LIN {X 0.262,Y -671.425,Z 418.419,A 0.000,B 0.000,C 90.000,E1 291.408} C_DIS
LIN {X -0.297,Y -673.117,Z 418.412,A 0.000,B 0.000,C 90.000,E1 290.248} C_DIS
LIN {X -0.129,Y -673.902,Z 418.407,A 0.000,B 0.000,C 90.000,E1 289.268} C_DIS
LIN {X -0.108,Y -674.468,Z 418.403,A 0.000,B 0.000,C 90.000,E1 288.544} C_DIS
LIN {X 0.005,Y -675.043,Z 418.396,A 0.000,B 0.000,C 90.000,E1 287.330} C_DIS
LIN {X -0.218,Y -675.211,Z 418.391,A 0.000,B 0.000,C 90.000,E1 286.386} C_DIS
LIN {X -0.297,Y -675.251,Z 418.384,A 0.000,B 0.000,C 90.000,E1 285.190} C_DIS
LIN {X 0.102,Y -675.047,Z 418.378,A 0.000,B 0.000,C 90.000,E1 283.953} C_DIS
LIN {X -0.211,Y -674.521,Z 418.370,A 0.000,B 0.000,C 90.000,E1 282.535} C_DIS
LIN {X -0.024,Y -673.626,Z 418.362,A 0.000,B 0.000,C 90.000,E1 281.074} C_DIS
LIN {X 0.207,Y -672.646,Z 418.355,A 0.000,B 0.000,C 90.000,E1 279.849} C_DIS
LIN {X 0.235,Y -671.359,Z 418.347,A 0.000,B 0.000,C 90.000,E1 278.398} C_DIS
LIN {X -0.033,Y -669.490,Z 418.336,A 0.000,B 0.000,C 90.000,E1 276.486} C_DIS
LIN {X -0.069,Y -668.227,Z 418.329,A 0.000,B 0.000,C 90.000,E1 275.277} C_DIS
LIN {X -0.176,Y -666.863,Z 418.323,A 0.000,B 0.000,C 90.000,E1 274.073} C_DIS
LIN {X -0.258,Y -665.172,Z 418.316,A 0.000,B 0.000,C 90.000,E1 272.865} C_DIS
LIN {X -0.263,Y -663.871,Z 418.310,A 0.000,B 0.000,C 90.000,E1 271.892} C_DIS
LIN {X 0.052,Y -661.562,Z 418.302,A 0.000,B 0.000,C 90.000,E1 270.401} C_DIS
LIN {X -0.174,Y -659.257,Z 418.296,A 0.000,B 0.000,C 90.000,E1 269.198} C_DIS
LIN {X 0.235,Y -656.673,Z 418.289,A 0.000,B 0.000,C 90.000,E1 267.936} C_DIS
LIN {X -0.252,Y -653.217,Z 418.280,A 0.000,B 0.000,C 90.000,E1 266.502} C_DIS
LIN {X -0.115,Y -649.497,Z 418.272,A 0.000,B 0.000,C 90.000,E1 265.008} C_DIS
LIN {X 0.172,Y -646.188,Z 418.265,A 0.000,B 0.000,C 90.000,E1 263.742} C_DIS
LIN {X -0.163,Y -642.674,Z 418.258,A 0.000,B 0.000,C 90.000,E1 262.527} C_DIS
LIN {X 0.085,Y -638.920,Z 418.251,A 0.000,B 0.000,C 90.000,E1 261.254} C_DIS
LIN {X 0.257,Y -635.010,Z 418.245,A 0.000,B 0.000,C 90.000,E1 259.982} C_DIS
LIN {X -0.157,Y -631.024,Z 418.238,A 0.000,B 0.000,C 90.000,E1 258.757} C_DIS
LIN {X 0.308,Y -627.809,Z 418.232,A 0.000,B 0.000,C 90.000,E1 257.701} C_DIS
LIN {X 0.311,Y -622.852,Z 418.223,A 0.000,B 0.000,C 90.000,E1 256.172} C_DIS
LIN {X 0.052,Y -619.414,Z 418.218,A 0.000,B 0.000,C 90.000,E1 255.172} C_DIS
LIN {X -0.325,Y -614.936,Z 418.211,A 0.000,B 0.000,C 90.000,E1 253.921} C_DIS
LIN {X -0.260,Y -609.408,Z 418.202,A 0.000,B 0.000,C 90.000,E1 252.362} C_DIS
LIN {X -0.042,Y -604.626,Z 418.195,A 0.000,B 0.000,C 90.000,E1 251.040} C_DIS
LIN {X 0.199,Y -598.715,Z 418.186,A 0.000,B 0.000,C 90.000,E1 249.444} C_DIS
LIN {X -0.036,Y -594.599,Z 418.180,A 0.000,B 0.000,C 90.000,E1 248.411} C_DIS
LIN {X -0.110,Y -590.373,Z 418.174,A 0.000,B 0.000,C 90.000,E1 247.358} C_DIS
LIN {X 0.174,Y -584.953,Z 418.167,A 0.000,B 0.000,C 90.000,E1 245.997} C_DIS
LIN {X 0.064,Y -579.379,Z 418.159,A 0.000,B 0.000,C 90.000,E1 244.665} C_DIS
LIN {X -0.191,Y -571.625,Z 418.149,A 0.000,B 0.000,C 90.000,E1 242.794} C_DIS
LIN {X 0.055,Y -564.970,Z 418.140,A 0.000,B 0.000,C 90.000,E1 241.129} C_DIS
LIN {X 0.206,Y -558.507,Z 418.130,A 0.000,B 0.000,C 90.000,E1 239.459} C_DIS
LIN {X 0.046,Y -550.141,Z 418.118,A 0.000,B 0.000,C 90.000,E1 237.248} C_DIS
LIN {X -0.278,Y -544.124,Z 418.109,A 0.000,B 0.000,C 90.000,E1 235.595} C_DIS
LIN {X 0.018,Y -538.215,Z 418.099,A 0.000,B 0.000,C 90.000,E1 233.863} C_DIS
LIN {X 0.059,Y -533.367,Z 418.091,A 0.000,B 0.000,C 90.000,E1 232.431} C_DIS
LIN {X -0.095,Y -527.441,Z 418.082,A 0.000,B 0.000,C 90.000,E1 230.723} C_DIS
LIN {X 0.096,Y -518.241,Z 418.066,A 0.000,B 0.000,C 90.000,E1 227.796} C_DIS
LIN {X 0.015,Y -513.892,Z 418.057,A 0.000,B 0.000,C 90.000,E1 226.338} C_DIS
LIN {X -0.240,Y -508.752,Z 418.048,A 0.000,B 0.000,C 90.000,E1 224.595} C_DIS
LIN {X 0.108,Y -503.657,Z 418.038,A 0.000,B 0.000,C 90.000,E1 222.771} C_DIS
LIN {X -0.137,Y -497.952,Z 418.026,A 0.000,B 0.000,C 90.000,E1 220.701} C_DIS
LIN {X -0.011,Y -493.110,Z 418.016,A 0.000,B 0.000,C 90.000,E1 218.874} C_DIS
LIN {X 0.156,Y -488.555,Z 418.006,A 0.000,B 0.000,C 90.000,E1 217.030} C_DIS
LIN {X -0.121,Y -482.585,Z 417.992,A 0.000,B 0.000,C 90.000,E1 214.612} C_DIS
LIN {X -0.060,Y -478.327,Z 417.982,A 0.000,B 0.000,C 90.000,E1 212.752} C_DIS
LIN {X -0.138,Y -474.780,Z 417.973,A 0.000,B 0.000,C 90.000,E1 211.209} C_DIS
LIN {X 0.056,Y -469.855,Z 417.961,A 0.000,B 0.000,C 90.000,E1 208.999} C_DIS
LIN {X -0.016,Y -466.300,Z 417.952,A 0.000,B 0.000,C 90.000,E1 207.436} C_DIS
LIN {X 0.095,Y -461.208,Z 417.940,A 0.000,B 0.000,C 90.000,E1 205.207} C_DIS
LIN {X -0.128,Y -457.419,Z 417.931,A 0.000,B 0.000,C 90.000,E1 203.643} C_DIS
LIN {X -0.101,Y -452.986,Z 417.921,A 0.000,B 0.000,C 90.000,E1 201.716} C_DIS
LIN {X 0.121,Y -446.616,Z 417.904,A 0.000,B 0.000,C 90.000,E1 198.779} C_DIS
LIN {X 0.117,Y -441.013,Z 417.888,A 0.000,B 0.000,C 90.000,E1 195.843} C_DIS
LIN {X 0.165,Y -437.031,Z 417.875,A 0.000,B 0.000,C 90.000,E1 193.536} C_DIS
LIN {X -0.001,Y -433.354,Z 417.863,A 0.000,B 0.000,C 90.000,E1 191.243} C_DIS
LIN {X -0.125,Y -430.451,Z 417.851,A 0.000,B 0.000,C 90.000,E1 189.265} C_DIS
LIN {X 0.041,Y -427.763,Z 417.840,A 0.000,B 0.000,C 90.000,E1 187.239} C_DIS
LIN {X 0.000,Y -425.763,Z 417.831,A 0.000,B 0.000,C 90.000,E1 185.568} C_DIS
LIN {X -0.082,Y -423.902,Z 417.822,A 0.000,B 0.000,C 90.000,E1 183.898} C_DIS
LIN {X -0.040,Y -420.972,Z 417.803,A 0.000,B 0.000,C 90.000,E1 180.516} C_DIS
LIN {X 0.039,Y -418.553,Z 417.776,A 0.000,B 0.000,C 90.000,E1 175.755} C_DIS
LIN {X 0.085,Y -418.119,Z 417.756,A 0.000,B 0.000,C 90.000,E1 172.008} C_DIS
LIN {X -0.051,Y -419.034,Z 417.735,A 0.000,B 0.000,C 90.000,E1 168.285} C_DIS
LIN {X 0.022,Y -421.832,Z 417.710,A 0.000,B 0.000,C 90.000,E1 163.866} C_DIS
LIN {X -0.028,Y -425.066,Z 417.692,A 0.000,B 0.000,C 90.000,E1 160.496} C_DIS
LIN {X -0.117,Y -428.740,Z 417.675,A 0.000,B 0.000,C 90.000,E1 157.486} C_DIS
LIN {X 0.048,Y -432.556,Z 417.660,A 0.000,B 0.000,C 90.000,E1 154.793} C_DIS
LIN {X -0.062,Y -437.123,Z 417.645,A 0.000,B 0.000,C 90.000,E1 152.153} C_DIS
LIN {X -0.251,Y -441.510,Z 417.632,A 0.000,B 0.000,C 90.000,E1 149.871} C_DIS
LIN {X -0.192,Y -447.154,Z 417.618,A 0.000,B 0.000,C 90.000,E1 147.248} C_DIS
LIN {X 0.171,Y -453.444,Z 417.604,A 0.000,B 0.000,C 90.000,E1 144.609} C_DIS
LIN {X 0.144,Y -462.963,Z 417.584,A 0.000,B 0.000,C 90.000,E1 141.090} C_DIS
LIN {X -0.089,Y -468.577,Z 417.573,A 0.000,B 0.000,C 90.000,E1 139.218} C_DIS
LIN {X 0.023,Y -473.242,Z 417.565,A 0.000,B 0.000,C 90.000,E1 137.634} C_DIS
LIN {X 0.190,Y -477.634,Z 417.556,A 0.000,B 0.000,C 90.000,E1 136.053} C_DIS
LIN {X 0.099,Y -481.585,Z 417.547,A 0.000,B 0.000,C 90.000,E1 134.514} C_DIS
LIN {X 0.076,Y -485.067,Z 417.539,A 0.000,B 0.000,C 90.000,E1 132.975} C_DIS
LIN {X -0.011,Y -487.422,Z 417.532,A 0.000,B 0.000,C 90.000,E1 131.757} C_DIS
LIN {X -0.061,Y -489.231,Z 417.525,A 0.000,B 0.000,C 90.000,E1 130.539} C_DIS
LIN {X -0.090,Y -490.238,Z 417.518,A 0.000,B 0.000,C 90.000,E1 129.322} C_DIS
LIN {X 0.121,Y -490.521,Z 417.513,A 0.000,B 0.000,C 90.000,E1 128.382} C_DIS
LIN {X -0.050,Y -490.146,Z 417.508,A 0.000,B 0.000,C 90.000,E1 127.488} C_DIS
LIN {X -0.134,Y -489.225,Z 417.503,A 0.000,B 0.000,C 90.000,E1 126.583} C_DIS
LIN {X 0.066,Y -488.011,Z 417.498,A 0.000,B 0.000,C 90.000,E1 125.644} C_DIS
LIN {X 0.133,Y -487.019,Z 417.495,A 0.000,B 0.000,C 90.000,E1 125.025} C_DIS
LIN {X 0.024,Y -485.155,Z 417.490,A 0.000,B 0.000,C 90.000,E1 124.119} C_DIS
LIN {X -0.110,Y -482.741,Z 417.484,A 0.000,B 0.000,C 90.000,E1 123.214} C_DIS
LIN {X -0.081,Y -480.984,Z 417.481,A 0.000,B 0.000,C 90.000,E1 122.594} C_DIS
LIN {X 0.086,Y -479.023,Z 417.478,A 0.000,B 0.000,C 90.000,E1 121.957} C_DIS
LIN {X -0.121,Y -475.839,Z 417.472,A 0.000,B 0.000,C 90.000,E1 121.052} C_DIS
LIN {X -0.027,Y -471.072,Z 417.466,A 0.000,B 0.000,C 90.000,E1 119.795} C_DIS
LIN {X -0.170,Y -467.241,Z 417.460,A 0.000,B 0.000,C 90.000,E1 118.871} C_DIS
LIN {X -0.030,Y -461.906,Z 417.453,A 0.000,B 0.000,C 90.000,E1 117.590} C_DIS
LIN {X -0.020,Y -455.619,Z 417.445,A 0.000,B 0.000,C 90.000,E1 116.155} C_DIS
LIN {X -0.109,Y -449.134,Z 417.437,A 0.000,B 0.000,C 90.000,E1 114.719} C_DIS
LIN {X -0.024,Y -446.480,Z 417.434,A 0.000,B 0.000,C 90.000,E1 114.131} C_DIS
LIN {X -0.064,Y -446.484,Z 417.434,A 0.000,B 0.000,C 90.000,E1 114.131} C_DIS
LIN {X 0.107,Y -455.340,Z 417.414,A 0.000,B 0.000,C 90.000,E1 110.482} C_DIS
LIN {X -0.097,Y -457.139,Z 417.410,A 0.000,B 0.000,C 90.000,E1 109.866} C_DIS
LIN {X 0.200,Y -466.537,Z 417.386,A 0.000,B 0.000,C 90.000,E1 105.371} C_DIS
LIN {X -0.074,Y -467.993,Z 417.382,A 0.000,B 0.000,C 90.000,E1 104.773} C_DIS
LIN {X -0.110,Y -476.209,Z 417.356,A 0.000,B 0.000,C 90.000,E1 100.074} C_DIS
LIN {X 0.145,Y -482.110,Z 417.330,A 0.000,B 0.000,C 90.000,E1 95.391} C_DIS
LIN {X -0.106,Y -485.518,Z 417.304,A 0.000,B 0.000,C 90.000,E1 90.802} C_DIS
LIN {X -0.073,Y -486.381,Z 417.281,A 0.000,B 0.000,C 90.000,E1 86.502} C_DIS
LIN {X -0.249,Y -486.357,Z 417.279,A 0.000,B 0.000,C 90.000,E1 86.216} C_DIS
LIN {X -0.165,Y -484.677,Z 417.253,A 0.000,B 0.000,C 90.000,E1 81.602} C_DIS
LIN {X 0.203,Y -480.595,Z 417.228,A 0.000,B 0.000,C 90.000,E1 76.937} C_DIS
LIN {X -0.083,Y -479.696,Z 417.224,A 0.000,B 0.000,C 90.000,E1 76.353} C_DIS
LIN {X -0.050,Y -474.039,Z 417.200,A 0.000,B 0.000,C 90.000,E1 72.000} C_DIS
LIN {X -0.207,Y -467.533,Z 417.180,A 0.000,B 0.000,C 90.000,E1 68.411} C_DIS
LIN {X -0.248,Y -467.542,Z 417.180,A 0.000,B 0.000,C 90.000,E1 68.411} C_DIS
LIN {X 0.240,Y -481.682,Z 417.170,A 0.000,B 0.000,C 90.000,E1 66.485} C_DIS
LIN {X -0.198,Y -488.819,Z 417.164,A 0.000,B 0.000,C 90.000,E1 65.613} C_DIS
LIN {X 0.052,Y -493.349,Z 417.161,A 0.000,B 0.000,C 90.000,E1 64.973} C_DIS
LIN {X -0.052,Y -499.831,Z 417.156,A 0.000,B 0.000,C 90.000,E1 64.076} C_DIS
LIN {X -0.122,Y -504.835,Z 417.152,A 0.000,B 0.000,C 90.000,E1 63.332} C_DIS
LIN {X 0.077,Y -509.514,Z 417.148,A 0.000,B 0.000,C 90.000,E1 62.564} C_DIS
LIN {X 0.223,Y -512.174,Z 417.145,A 0.000,B 0.000,C 90.000,E1 62.103} C_DIS
LIN {X 0.041,Y -516.129,Z 417.141,A 0.000,B 0.000,C 90.000,E1 61.385} C_DIS
LIN {X 0.060,Y -519.050,Z 417.138,A 0.000,B 0.000,C 90.000,E1 60.795} C_DIS
LIN {X 0.101,Y -521.660,Z 417.135,A 0.000,B 0.000,C 90.000,E1 60.205} C_DIS
LIN {X -0.131,Y -523.451,Z 417.132,A 0.000,B 0.000,C 90.000,E1 59.793} C_DIS
LIN {X -0.110,Y -526.612,Z 417.127,A 0.000,B 0.000,C 90.000,E1 58.918} C_DIS
LIN {X -0.019,Y -528.342,Z 417.124,A 0.000,B 0.000,C 90.000,E1 58.329} C_DIS
LIN {X 0.052,Y -530.398,Z 417.119,A 0.000,B 0.000,C 90.000,E1 57.454} C_DIS
LIN {X -0.282,Y -531.505,Z 417.116,A 0.000,B 0.000,C 90.000,E1 56.914} C_DIS
LIN {X 0.112,Y -532.629,Z 417.111,A 0.000,B 0.000,C 90.000,E1 56.008} C_DIS
LIN {X -0.209,Y -533.125,Z 417.108,A 0.000,B 0.000,C 90.000,E1 55.468} C_DIS
LIN {X 0.205,Y -533.431,Z 417.103,A 0.000,B 0.000,C 90.000,E1 54.562} C_DIS
LIN {X 0.189,Y -533.448,Z 417.099,A 0.000,B 0.000,C 90.000,E1 53.703} C_DIS
LIN {X 0.176,Y -533.149,Z 417.094,A 0.000,B 0.000,C 90.000,E1 52.844} C_DIS
LIN {X 0.150,Y -532.380,Z 417.087,A 0.000,B 0.000,C 90.000,E1 51.698} C_DIS
LIN {X 0.029,Y -531.319,Z 417.081,A 0.000,B 0.000,C 90.000,E1 50.561} C_DIS
LIN {X 0.306,Y -530.052,Z 417.075,A 0.000,B 0.000,C 90.000,E1 49.380} C_DIS
LIN {X 0.157,Y -528.545,Z 417.068,A 0.000,B 0.000,C 90.000,E1 48.243} C_DIS
LIN {X -0.087,Y -526.474,Z 417.060,A 0.000,B 0.000,C 90.000,E1 46.824} C_DIS
LIN {X -0.181,Y -523.226,Z 417.047,A 0.000,B 0.000,C 90.000,E1 44.514} C_DIS
LIN {X 0.012,Y -520.378,Z 417.034,A 0.000,B 0.000,C 90.000,E1 42.162} C_DIS
LIN {X 0.010,Y -518.615,Z 417.026,A 0.000,B 0.000,C 90.000,E1 40.701} C_DIS
LIN {X -0.037,Y -516.925,Z 417.018,A 0.000,B 0.000,C 90.000,E1 39.241} C_DIS
LIN {X -0.301,Y -515.616,Z 417.012,A 0.000,B 0.000,C 90.000,E1 38.096} C_DIS
LIN {X 0.000,Y -513.495,Z 417.002,A 0.000,B 0.000,C 90.000,E1 36.297} C_DIS
LIN {X 0.028,Y -511.646,Z 416.993,A 0.000,B 0.000,C 90.000,E1 34.818} C_DIS
LIN {X -0.266,Y -509.717,Z 416.985,A 0.000,B 0.000,C 90.000,E1 33.372} C_DIS
LIN {X -0.319,Y -506.507,Z 416.972,A 0.000,B 0.000,C 90.000,E1 31.003} C_DIS
LIN {X 0.077,Y -503.697,Z 416.960,A 0.000,B 0.000,C 90.000,E1 28.871} C_DIS
LIN {X -0.098,Y -501.106,Z 416.949,A 0.000,B 0.000,C 90.000,E1 26.796} C_DIS
LIN {X -0.057,Y -498.400,Z 416.935,A 0.000,B 0.000,C 90.000,E1 24.387} C_DIS
LIN {X -0.035,Y -496.137,Z 416.922,A 0.000,B 0.000,C 90.000,E1 21.972} C_DIS
LIN {X -0.161,Y -493.871,Z 416.905,A 0.000,B 0.000,C 90.000,E1 18.960} C_DIS
LIN {X 0.232,Y -492.610,Z 416.895,A 0.000,B 0.000,C 90.000,E1 17.094} C_DIS
LIN {X -0.043,Y -491.588,Z 416.887,A 0.000,B 0.000,C 90.000,E1 15.607} C_DIS
LIN {X 0.032,Y -490.431,Z 416.877,A 0.000,B 0.000,C 90.000,E1 13.772} C_DIS
LIN {X -0.252,Y -489.257,Z 416.863,A 0.000,B 0.000,C 90.000,E1 11.366} C_DIS
LIN {X 0.057,Y -488.469,Z 416.846,A 0.000,B 0.000,C 90.000,E1 8.276} C_DIS
LIN {X 0.178,Y -488.364,Z 416.831,A 0.000,B 0.000,C 90.000,E1 5.511} C_DIS
LIN {X -0.224,Y -489.458,Z 416.810,A 0.000,B 0.000,C 90.000,E1 1.892} C_DIS
LIN {X -0.194,Y -493.605,Z 416.784,A 0.000,B 0.000,C 90.000,E1 357.078} C_DIS
LIN {X -0.041,Y -495.895,Z 416.774,A 0.000,B 0.000,C 90.000,E1 355.241} C_DIS
LIN {X -0.056,Y -499.914,Z 416.758,A 0.000,B 0.000,C 90.000,E1 352.527} C_DIS
LIN {X 0.037,Y -505.631,Z 416.740,A 0.000,B 0.000,C 90.000,E1 349.218} C_DIS
LIN {X 0.156,Y -512.535,Z 416.722,A 0.000,B 0.000,C 90.000,E1 345.936} C_DIS
LIN {X 0.132,Y -516.072,Z 416.714,A 0.000,B 0.000,C 90.000,E1 344.464} C_DIS
LIN {X -0.062,Y -520.476,Z 416.704,A 0.000,B 0.000,C 90.000,E1 342.725} C_DIS
LIN {X -0.002,Y -525.767,Z 416.693,A 0.000,B 0.000,C 90.000,E1 340.678} C_DIS
LIN {X 0.054,Y -532.197,Z 416.680,A 0.000,B 0.000,C 90.000,E1 338.358} C_DIS
LIN {X -0.011,Y -537.896,Z 416.669,A 0.000,B 0.000,C 90.000,E1 336.357} C_DIS
LIN {X -0.160,Y -542.870,Z 416.659,A 0.000,B 0.000,C 90.000,E1 334.665} C_DIS
LIN {X 0.024,Y -548.000,Z 416.650,A 0.000,B 0.000,C 90.000,E1 332.948} C_DIS
LIN {X 0.121,Y -554.214,Z 416.639,A 0.000,B 0.000,C 90.000,E1 330.973} C_DIS
LIN {X -0.164,Y -559.600,Z 416.630,A 0.000,B 0.000,C 90.000,E1 329.331} C_DIS
LIN {X -0.060,Y -564.899,Z 416.620,A 0.000,B 0.000,C 90.000,E1 327.661} C_DIS
LIN {X -0.138,Y -569.258,Z 416.613,A 0.000,B 0.000,C 90.000,E1 326.294} C_DIS
LIN {X -0.010,Y -574.495,Z 416.604,A 0.000,B 0.000,C 90.000,E1 324.642} C_DIS
LIN {X -0.208,Y -580.640,Z 416.593,A 0.000,B 0.000,C 90.000,E1 322.763} C_DIS
LIN {X -0.064,Y -587.860,Z 416.581,A 0.000,B 0.000,C 90.000,E1 320.598} C_DIS
LIN {X -0.026,Y -594.350,Z 416.571,A 0.000,B 0.000,C 90.000,E1 318.728} C_DIS
LIN {X 0.115,Y -600.693,Z 416.560,A 0.000,B 0.000,C 90.000,E1 316.863} C_DIS
LIN {X -0.263,Y -606.157,Z 416.552,A 0.000,B 0.000,C 90.000,E1 315.324} C_DIS
LIN {X 0.336,Y -611.680,Z 416.543,A 0.000,B 0.000,C 90.000,E1 313.704} C_DIS
LIN {X -0.083,Y -616.262,Z 416.536,A 0.000,B 0.000,C 90.000,E1 312.447} C_DIS
LIN {X -0.123,Y -621.803,Z 416.527,A 0.000,B 0.000,C 90.000,E1 310.906} C_DIS
LIN {X -0.176,Y -625.335,Z 416.522,A 0.000,B 0.000,C 90.000,E1 309.886} C_DIS
LIN {X 0.223,Y -628.748,Z 416.516,A 0.000,B 0.000,C 90.000,E1 308.830} C_DIS
LIN {X -0.247,Y -632.916,Z 416.509,A 0.000,B 0.000,C 90.000,E1 307.604} C_DIS
LIN {X 0.238,Y -636.875,Z 416.502,A 0.000,B 0.000,C 90.000,E1 306.297} C_DIS
LIN {X 0.012,Y -639.944,Z 416.496,A 0.000,B 0.000,C 90.000,E1 305.311} C_DIS
LIN {X -0.174,Y -642.928,Z 416.491,A 0.000,B 0.000,C 90.000,E1 304.326} C_DIS
LIN {X -0.274,Y -646.585,Z 416.484,A 0.000,B 0.000,C 90.000,E1 303.086} C_DIS
LIN {X -0.153,Y -651.558,Z 416.474,A 0.000,B 0.000,C 90.000,E1 301.337} C_DIS
LIN {X -0.356,Y -655.583,Z 416.466,A 0.000,B 0.000,C 90.000,E1 299.873} C_DIS
LIN {X 0.304,Y -657.493,Z 416.462,A 0.000,B 0.000,C 90.000,E1 299.077} C_DIS
LIN {X 0.214,Y -659.915,Z 416.456,A 0.000,B 0.000,C 90.000,E1 298.103} C_DIS
LIN {X -0.163,Y -663.392,Z 416.448,A 0.000,B 0.000,C 90.000,E1 296.668} C_DIS
LIN {X 0.269,Y -666.125,Z 416.441,A 0.000,B 0.000,C 90.000,E1 295.412} C_DIS
LIN {X -0.161,Y -667.744,Z 416.437,A 0.000,B 0.000,C 90.000,E1 294.719} C_DIS
LIN {X -0.418,Y -669.625,Z 416.432,A 0.000,B 0.000,C 90.000,E1 293.770} C_DIS
LIN {X -0.040,Y -671.367,Z 416.427,A 0.000,B 0.000,C 90.000,E1 292.770} C_DIS
LIN {X 0.106,Y -672.878,Z 416.421,A 0.000,B 0.000,C 90.000,E1 291.791} C_DIS
LIN {X -0.187,Y -674.540,Z 416.414,A 0.000,B 0.000,C 90.000,E1 290.610} C_DIS
LIN {X -0.163,Y -675.238,Z 416.410,A 0.000,B 0.000,C 90.000,E1 289.885} C_DIS
LIN {X -0.026,Y -675.994,Z 416.404,A 0.000,B 0.000,C 90.000,E1 288.671} C_DIS
LIN {X 0.170,Y -676.335,Z 416.398,A 0.000,B 0.000,C 90.000,E1 287.692} C_DIS
LIN {X 0.157,Y -676.467,Z 416.393,A 0.000,B 0.000,C 90.000,E1 286.732} C_DIS
LIN {X -0.043,Y -676.406,Z 416.388,A 0.000,B 0.000,C 90.000,E1 285.788} C_DIS
LIN {X -0.010,Y -676.281,Z 416.384,A 0.000,B 0.000,C 90.000,E1 285.064} C_DIS
LIN {X -0.208,Y -675.998,Z 416.378,A 0.000,B 0.000,C 90.000,E1 284.120} C_DIS
LIN {X 0.093,Y -675.159,Z 416.369,A 0.000,B 0.000,C 90.000,E1 282.411} C_DIS
LIN {X 0.281,Y -674.212,Z 416.361,A 0.000,B 0.000,C 90.000,E1 280.950} C_DIS
LIN {X -0.330,Y -672.998,Z 416.353,A 0.000,B 0.000,C 90.000,E1 279.557} C_DIS
LIN {X -0.298,Y -671.680,Z 416.345,A 0.000,B 0.000,C 90.000,E1 278.106} C_DIS
LIN {X 0.027,Y -669.804,Z 416.334,A 0.000,B 0.000,C 90.000,E1 276.144} C_DIS
LIN {X 0.004,Y -668.480,Z 416.327,A 0.000,B 0.000,C 90.000,E1 274.935} C_DIS
LIN {X 0.118,Y -667.377,Z 416.322,A 0.000,B 0.000,C 90.000,E1 273.955} C_DIS
LIN {X -0.001,Y -665.674,Z 416.315,A 0.000,B 0.000,C 90.000,E1 272.751} C_DIS
LIN {X 0.021,Y -664.414,Z 416.310,A 0.000,B 0.000,C 90.000,E1 271.776} C_DIS
LIN {X 0.327,Y -662.212,Z 416.302,A 0.000,B 0.000,C 90.000,E1 270.286} C_DIS
LIN {X 0.288,Y -660.497,Z 416.296,A 0.000,B 0.000,C 90.000,E1 269.312} C_DIS
LIN {X 0.059,Y -658.130,Z 416.290,A 0.000,B 0.000,C 90.000,E1 268.108} C_DIS
LIN {X -0.235,Y -655.415,Z 416.283,A 0.000,B 0.000,C 90.000,E1 266.906} C_DIS
LIN {X 0.146,Y -652.540,Z 416.276,A 0.000,B 0.000,C 90.000,E1 265.641} C_DIS
LIN {X -0.003,Y -650.058,Z 416.270,A 0.000,B 0.000,C 90.000,E1 264.666} C_DIS
LIN {X -0.125,Y -647.441,Z 416.265,A 0.000,B 0.000,C 90.000,E1 263.685} C_DIS
LIN {X 0.198,Y -643.943,Z 416.258,A 0.000,B 0.000,C 90.000,E1 262.413} C_DIS
LIN {X -0.171,Y -640.235,Z 416.251,A 0.000,B 0.000,C 90.000,E1 261.197} C_DIS
LIN {X 0.022,Y -636.355,Z 416.244,A 0.000,B 0.000,C 90.000,E1 259.926} C_DIS
LIN {X -0.371,Y -632.399,Z 416.237,A 0.000,B 0.000,C 90.000,E1 258.701} C_DIS
LIN {X 0.112,Y -629.168,Z 416.231,A 0.000,B 0.000,C 90.000,E1 257.645} C_DIS
LIN {X 0.139,Y -624.218,Z 416.223,A 0.000,B 0.000,C 90.000,E1 256.117} C_DIS
LIN {X -0.160,Y -619.895,Z 416.216,A 0.000,B 0.000,C 90.000,E1 254.866} C_DIS
LIN {X 0.071,Y -615.362,Z 416.209,A 0.000,B 0.000,C 90.000,E1 253.559} C_DIS
LIN {X -0.372,Y -610.749,Z 416.202,A 0.000,B 0.000,C 90.000,E1 252.308} C_DIS
LIN {X 0.062,Y -605.961,Z 416.194,A 0.000,B 0.000,C 90.000,E1 250.967} C_DIS
LIN {X 0.128,Y -599.994,Z 416.186,A 0.000,B 0.000,C 90.000,E1 249.390} C_DIS
LIN {X 0.127,Y -595.875,Z 416.180,A 0.000,B 0.000,C 90.000,E1 248.337} C_DIS
LIN {X -0.255,Y -590.546,Z 416.172,A 0.000,B 0.000,C 90.000,E1 247.050} C_DIS
LIN {X 0.269,Y -585.087,Z 416.165,A 0.000,B 0.000,C 90.000,E1 245.665} C_DIS
LIN {X 0.170,Y -579.483,Z 416.158,A 0.000,B 0.000,C 90.000,E1 244.332} C_DIS
LIN {X -0.180,Y -572.823,Z 416.149,A 0.000,B 0.000,C 90.000,E1 242.743} C_DIS
LIN {X -0.138,Y -566.185,Z 416.139,A 0.000,B 0.000,C 90.000,E1 241.101} C_DIS
LIN {X 0.045,Y -558.654,Z 416.129,A 0.000,B 0.000,C 90.000,E1 239.154} C_DIS
LIN {X 0.170,Y -550.346,Z 416.116,A 0.000,B 0.000,C 90.000,E1 236.914} C_DIS
LIN {X -0.154,Y -544.391,Z 416.107,A 0.000,B 0.000,C 90.000,E1 235.261} C_DIS
LIN {X 0.023,Y -538.493,Z 416.098,A 0.000,B 0.000,C 90.000,E1 233.543} C_DIS
LIN {X 0.076,Y -534.625,Z 416.091,A 0.000,B 0.000,C 90.000,E1 232.396} C_DIS
LIN {X 0.036,Y -528.739,Z 416.082,A 0.000,B 0.000,C 90.000,E1 230.678} C_DIS
LIN {X -0.131,Y -519.531,Z 416.065,A 0.000,B 0.000,C 90.000,E1 227.796} C_DIS
LIN {X -0.271,Y -514.279,Z 416.056,A 0.000,B 0.000,C 90.000,E1 226.053} C_DIS
LIN {X -0.055,Y -510.018,Z 416.048,A 0.000,B 0.000,C 90.000,E1 224.555} C_DIS
LIN {X 0.192,Y -504.075,Z 416.036,A 0.000,B 0.000,C 90.000,E1 222.447} C_DIS
LIN {X -0.049,Y -498.394,Z 416.024,A 0.000,B 0.000,C 90.000,E1 220.378} C_DIS
LIN {X 0.010,Y -492.787,Z 416.013,A 0.000,B 0.000,C 90.000,E1 218.257} C_DIS
LIN {X -0.048,Y -489.014,Z 416.004,A 0.000,B 0.000,C 90.000,E1 216.744} C_DIS
LIN {X -0.134,Y -483.810,Z 415.992,A 0.000,B 0.000,C 90.000,E1 214.612} C_DIS
LIN {X 0.160,Y -478.825,Z 415.980,A 0.000,B 0.000,C 90.000,E1 212.418} C_DIS
LIN {X -0.101,Y -475.977,Z 415.973,A 0.000,B 0.000,C 90.000,E1 211.209} C_DIS
LIN {X -0.047,Y -471.744,Z 415.963,A 0.000,B 0.000,C 90.000,E1 209.333} C_DIS
LIN {X -0.140,Y -467.472,Z 415.953,A 0.000,B 0.000,C 90.000,E1 207.462} C_DIS
LIN {X 0.091,Y -463.101,Z 415.942,A 0.000,B 0.000,C 90.000,E1 205.540} C_DIS
LIN {X 0.179,Y -460.116,Z 415.935,A 0.000,B 0.000,C 90.000,E1 204.259} C_DIS
LIN {X 0.164,Y -454.823,Z 415.923,A 0.000,B 0.000,C 90.000,E1 202.025} C_DIS
LIN {X 0.071,Y -451.151,Z 415.914,A 0.000,B 0.000,C 90.000,E1 200.429} C_DIS
LIN {X -0.075,Y -446.354,Z 415.901,A 0.000,B 0.000,C 90.000,E1 198.181} C_DIS
LIN {X -0.069,Y -442.054,Z 415.888,A 0.000,B 0.000,C 90.000,E1 195.898} C_DIS
LIN {X 0.005,Y -438.056,Z 415.876,A 0.000,B 0.000,C 90.000,E1 193.592} C_DIS
LIN {X -0.136,Y -434.347,Z 415.863,A 0.000,B 0.000,C 90.000,E1 191.299} C_DIS
LIN {X -0.123,Y -430.919,Z 415.850,A 0.000,B 0.000,C 90.000,E1 188.973} C_DIS
LIN {X -0.053,Y -428.688,Z 415.841,A 0.000,B 0.000,C 90.000,E1 187.296} C_DIS
LIN {X -0.075,Y -426.677,Z 415.831,A 0.000,B 0.000,C 90.000,E1 185.625} C_DIS
LIN {X 0.028,Y -423.813,Z 415.816,A 0.000,B 0.000,C 90.000,E1 182.922} C_DIS
LIN {X 0.059,Y -421.086,Z 415.798,A 0.000,B 0.000,C 90.000,E1 179.542} C_DIS
LIN {X 0.144,Y -419.196,Z 415.773,A 0.000,B 0.000,C 90.000,E1 175.122} C_DIS
LIN {X 0.083,Y -418.903,Z 415.758,A 0.000,B 0.000,C 90.000,E1 172.413} C_DIS
LIN {X 0.049,Y -419.798,Z 415.735,A 0.000,B 0.000,C 90.000,E1 168.342} C_DIS
LIN {X -0.066,Y -422.009,Z 415.715,A 0.000,B 0.000,C 90.000,E1 164.629} C_DIS
LIN {X -0.198,Y -424.384,Z 415.700,A 0.000,B 0.000,C 90.000,E1 161.945} C_DIS
LIN {X 0.140,Y -427.335,Z 415.685,A 0.000,B 0.000,C 90.000,E1 159.209} C_DIS
LIN {X 0.117,Y -430.377,Z 415.672,A 0.000,B 0.000,C 90.000,E1 156.869} C_DIS
LIN {X 0.128,Y -434.393,Z 415.657,A 0.000,B 0.000,C 90.000,E1 154.204} C_DIS
LIN {X 0.055,Y -438.475,Z 415.644,A 0.000,B 0.000,C 90.000,E1 151.897} C_DIS
LIN {X 0.119,Y -445.779,Z 415.624,A 0.000,B 0.000,C 90.000,E1 148.280} C_DIS
LIN {X -0.113,Y -452.642,Z 415.608,A 0.000,B 0.000,C 90.000,E1 145.388} C_DIS
LIN {X 0.037,Y -455.172,Z 415.602,A 0.000,B 0.000,C 90.000,E1 144.402} C_DIS
LIN {X 0.077,Y -464.883,Z 415.583,A 0.000,B 0.000,C 90.000,E1 140.884} C_DIS
LIN {X -0.118,Y -470.600,Z 415.572,A 0.000,B 0.000,C 90.000,E1 139.013} C_DIS
LIN {X -0.099,Y -474.367,Z 415.565,A 0.000,B 0.000,C 90.000,E1 137.757} C_DIS
LIN {X -0.234,Y -478.815,Z 415.557,A 0.000,B 0.000,C 90.000,E1 136.215} C_DIS
LIN {X 0.248,Y -482.108,Z 415.550,A 0.000,B 0.000,C 90.000,E1 134.919} C_DIS
LIN {X -0.038,Y -484.340,Z 415.545,A 0.000,B 0.000,C 90.000,E1 134.028} C_DIS
LIN {X 0.051,Y -486.434,Z 415.539,A 0.000,B 0.000,C 90.000,E1 133.095} C_DIS
LIN {X 0.166,Y -488.257,Z 415.534,A 0.000,B 0.000,C 90.000,E1 132.162} C_DIS
LIN {X -0.220,Y -489.412,Z 415.531,A 0.000,B 0.000,C 90.000,E1 131.595} C_DIS
LIN {X 0.131,Y -491.119,Z 415.524,A 0.000,B 0.000,C 90.000,E1 130.334} C_DIS
LIN {X 0.134,Y -492.111,Z 415.517,A 0.000,B 0.000,C 90.000,E1 129.116} C_DIS
LIN {X -0.016,Y -492.326,Z 415.512,A 0.000,B 0.000,C 90.000,E1 128.222} C_DIS
LIN {X -0.077,Y -491.918,Z 415.507,A 0.000,B 0.000,C 90.000,E1 127.317} C_DIS
LIN {X 0.159,Y -490.937,Z 415.502,A 0.000,B 0.000,C 90.000,E1 126.377} C_DIS
LIN {X -0.148,Y -490.155,Z 415.499,A 0.000,B 0.000,C 90.000,E1 125.804} C_DIS
LIN {X -0.221,Y -488.660,Z 415.494,A 0.000,B 0.000,C 90.000,E1 124.898} C_DIS
LIN {X -0.310,Y -486.746,Z 415.489,A 0.000,B 0.000,C 90.000,E1 123.992} C_DIS
LIN {X -0.016,Y -484.273,Z 415.484,A 0.000,B 0.000,C 90.000,E1 123.038} C_DIS
LIN {X 0.029,Y -482.483,Z 415.480,A 0.000,B 0.000,C 90.000,E1 122.418} C_DIS
LIN {X 0.269,Y -479.433,Z 415.475,A 0.000,B 0.000,C 90.000,E1 121.465} C_DIS
LIN {X 0.025,Y -477.234,Z 415.472,A 0.000,B 0.000,C 90.000,E1 120.875} C_DIS
LIN {X 0.145,Y -472.392,Z 415.465,A 0.000,B 0.000,C 90.000,E1 119.617} C_DIS
LIN {X 0.021,Y -468.514,Z 415.459,A 0.000,B 0.000,C 90.000,E1 118.693} C_DIS
LIN {X 0.015,Y -463.820,Z 415.453,A 0.000,B 0.000,C 90.000,E1 117.590} C_DIS
LIN {X 0.106,Y -458.195,Z 415.446,A 0.000,B 0.000,C 90.000,E1 116.309} C_DIS
LIN {X -0.152,Y -451.663,Z 415.438,A 0.000,B 0.000,C 90.000,E1 114.899} C_DIS
LIN {X -0.184,Y -447.026,Z 415.433,A 0.000,B 0.000,C 90.000,E1 113.898} C_DIS
LIN {X -0.222,Y -447.031,Z 415.433,A 0.000,B 0.000,C 90.000,E1 113.898} C_DIS
LIN {X -0.025,Y -455.737,Z 415.413,A 0.000,B 0.000,C 90.000,E1 110.355} C_DIS
LIN {X 0.048,Y -457.451,Z 415.410,A 0.000,B 0.000,C 90.000,E1 109.704} C_DIS
LIN {X 0.149,Y -466.110,Z 415.387,A 0.000,B 0.000,C 90.000,E1 105.552} C_DIS
LIN {X -0.127,Y -467.680,Z 415.383,A 0.000,B 0.000,C 90.000,E1 104.954} C_DIS
LIN {X -0.169,Y -475.893,Z 415.357,A 0.000,B 0.000,C 90.000,E1 100.254} C_DIS
LIN {X 0.138,Y -476.346,Z 415.355,A 0.000,B 0.000,C 90.000,E1 99.905} C_DIS
LIN {X 0.094,Y -481.859,Z 415.331,A 0.000,B 0.000,C 90.000,E1 95.568} C_DIS
LIN {X -0.059,Y -482.189,Z 415.329,A 0.000,B 0.000,C 90.000,E1 95.277} C_DIS
LIN {X -0.125,Y -485.354,Z 415.305,A 0.000,B 0.000,C 90.000,E1 90.974} C_DIS
LIN {X 0.185,Y -485.532,Z 415.304,A 0.000,B 0.000,C 90.000,E1 90.630} C_DIS
LIN {X -0.092,Y -486.341,Z 415.282,A 0.000,B 0.000,C 90.000,E1 86.674} C_DIS
LIN {X 0.041,Y -486.274,Z 415.278,A 0.000,B 0.000,C 90.000,E1 86.045} C_DIS
LIN {X -0.238,Y -484.694,Z 415.254,A 0.000,B 0.000,C 90.000,E1 81.781} C_DIS
LIN {X 0.109,Y -484.547,Z 415.253,A 0.000,B 0.000,C 90.000,E1 81.432} C_DIS
LIN {X -0.021,Y -480.486,Z 415.227,A 0.000,B 0.000,C 90.000,E1 76.825} C_DIS
LIN {X -0.124,Y -474.242,Z 415.201,A 0.000,B 0.000,C 90.000,E1 72.181} C_DIS
LIN {X -0.157,Y -473.756,Z 415.199,A 0.000,B 0.000,C 90.000,E1 71.873} C_DIS
LIN {X 0.096,Y -467.868,Z 415.181,A 0.000,B 0.000,C 90.000,E1 68.592} C_DIS
LIN {X 0.056,Y -467.895,Z 415.181,A 0.000,B 0.000,C 90.000,E1 68.592} C_DIS
LIN {X 0.073,Y -475.198,Z 415.176,A 0.000,B 0.000,C 90.000,E1 67.614} C_DIS
LIN {X -0.026,Y -486.030,Z 415.168,A 0.000,B 0.000,C 90.000,E1 66.230} C_DIS
LIN {X 0.026,Y -492.951,Z 415.163,A 0.000,B 0.000,C 90.000,E1 65.305} C_DIS
LIN {X -0.088,Y -499.479,Z 415.158,A 0.000,B 0.000,C 90.000,E1 64.409} C_DIS
LIN {X 0.252,Y -503.578,Z 415.154,A 0.000,B 0.000,C 90.000,E1 63.768} C_DIS
LIN {X 0.263,Y -509.321,Z 415.150,A 0.000,B 0.000,C 90.000,E1 62.871} C_DIS
LIN {X 0.057,Y -513.740,Z 415.145,A 0.000,B 0.000,C 90.000,E1 62.153} C_DIS
LIN {X 0.061,Y -516.911,Z 415.142,A 0.000,B 0.000,C 90.000,E1 61.563} C_DIS
LIN {X 0.088,Y -519.856,Z 415.139,A 0.000,B 0.000,C 90.000,E1 60.973} C_DIS
LIN {X -0.025,Y -523.073,Z 415.135,A 0.000,B 0.000,C 90.000,E1 60.255} C_DIS
LIN {X 0.045,Y -525.407,Z 415.132,A 0.000,B 0.000,C 90.000,E1 59.665} C_DIS
LIN {X 0.127,Y -527.496,Z 415.128,A 0.000,B 0.000,C 90.000,E1 59.076} C_DIS
LIN {X -0.228,Y -529.259,Z 415.125,A 0.000,B 0.000,C 90.000,E1 58.535} C_DIS
LIN {X -0.148,Y -531.419,Z 415.120,A 0.000,B 0.000,C 90.000,E1 57.661} C_DIS
LIN {X 0.259,Y -532.509,Z 415.117,A 0.000,B 0.000,C 90.000,E1 57.041} C_DIS
LIN {X -0.071,Y -533.750,Z 415.112,A 0.000,B 0.000,C 90.000,E1 56.215} C_DIS
LIN {X 0.050,Y -534.499,Z 415.108,A 0.000,B 0.000,C 90.000,E1 55.341} C_DIS
LIN {X 0.042,Y -534.705,Z 415.103,A 0.000,B 0.000,C 90.000,E1 54.482} C_DIS
LIN {X 0.042,Y -534.670,Z 415.098,A 0.000,B 0.000,C 90.000,E1 53.623} C_DIS
LIN {X 0.044,Y -534.332,Z 415.093,A 0.000,B 0.000,C 90.000,E1 52.763} C_DIS
LIN {X 0.040,Y -533.744,Z 415.088,A 0.000,B 0.000,C 90.000,E1 51.904} C_DIS
LIN {X 0.016,Y -532.660,Z 415.082,A 0.000,B 0.000,C 90.000,E1 50.759} C_DIS
LIN {X -0.102,Y -531.446,Z 415.076,A 0.000,B 0.000,C 90.000,E1 49.622} C_DIS
LIN {X 0.119,Y -529.975,Z 415.069,A 0.000,B 0.000,C 90.000,E1 48.447} C_DIS
LIN {X -0.066,Y -527.883,Z 415.061,A 0.000,B 0.000,C 90.000,E1 47.025} C_DIS
LIN {X 0.236,Y -524.576,Z 415.048,A 0.000,B 0.000,C 90.000,E1 44.676} C_DIS
LIN {X 0.226,Y -522.339,Z 415.039,A 0.000,B 0.000,C 90.000,E1 42.933} C_DIS
LIN {X -0.130,Y -520.622,Z 415.031,A 0.000,B 0.000,C 90.000,E1 41.515} C_DIS
LIN {X 0.141,Y -518.196,Z 415.019,A 0.000,B 0.000,C 90.000,E1 39.439} C_DIS
LIN {X -0.245,Y -516.504,Z 415.011,A 0.000,B 0.000,C 90.000,E1 38.016} C_DIS
LIN {X 0.144,Y -514.758,Z 415.003,A 0.000,B 0.000,C 90.000,E1 36.503} C_DIS
LIN {X 0.115,Y -512.514,Z 414.993,A 0.000,B 0.000,C 90.000,E1 34.739} C_DIS
LIN {X -0.080,Y -510.979,Z 414.987,A 0.000,B 0.000,C 90.000,E1 33.579} C_DIS
LIN {X -0.292,Y -509.306,Z 414.980,A 0.000,B 0.000,C 90.000,E1 32.418} C_DIS
LIN {X -0.204,Y -507.383,Z 414.972,A 0.000,B 0.000,C 90.000,E1 30.924} C_DIS
LIN {X -0.035,Y -504.590,Z 414.960,A 0.000,B 0.000,C 90.000,E1 28.821} C_DIS
LIN {X 0.201,Y -502.358,Z 414.950,A 0.000,B 0.000,C 90.000,E1 27.001} C_DIS
LIN {X -0.168,Y -499.662,Z 414.937,A 0.000,B 0.000,C 90.000,E1 24.643} C_DIS
LIN {X 0.085,Y -497.312,Z 414.923,A 0.000,B 0.000,C 90.000,E1 22.206} C_DIS
LIN {X -0.174,Y -495.002,Z 414.907,A 0.000,B 0.000,C 90.000,E1 19.214} C_DIS
LIN {X -0.105,Y -493.971,Z 414.898,A 0.000,B 0.000,C 90.000,E1 17.692} C_DIS
LIN {X 0.117,Y -492.918,Z 414.890,A 0.000,B 0.000,C 90.000,E1 16.150} C_DIS
LIN {X -0.126,Y -491.732,Z 414.880,A 0.000,B 0.000,C 90.000,E1 14.356} C_DIS
LIN {X 0.100,Y -490.482,Z 414.866,A 0.000,B 0.000,C 90.000,E1 11.895} C_DIS
LIN {X 0.096,Y -489.623,Z 414.851,A 0.000,B 0.000,C 90.000,E1 9.151} C_DIS
LIN {X -0.175,Y -489.423,Z 414.841,A 0.000,B 0.000,C 90.000,E1 7.352} C_DIS
LIN {X 0.206,Y -489.391,Z 414.834,A 0.000,B 0.000,C 90.000,E1 6.087} C_DIS
LIN {X 0.197,Y -490.051,Z 414.817,A 0.000,B 0.000,C 90.000,E1 3.037} C_DIS
LIN {X -0.008,Y -494.422,Z 414.785,A 0.000,B 0.000,C 90.000,E1 357.364} C_DIS
LIN {X -0.181,Y -496.302,Z 414.777,A 0.000,B 0.000,C 90.000,E1 355.869} C_DIS
LIN {X 0.130,Y -500.658,Z 414.760,A 0.000,B 0.000,C 90.000,E1 352.818} C_DIS
LIN {X 0.249,Y -506.291,Z 414.742,A 0.000,B 0.000,C 90.000,E1 349.511} C_DIS
LIN {X -0.033,Y -509.859,Z 414.732,A 0.000,B 0.000,C 90.000,E1 347.757} C_DIS
LIN {X -0.080,Y -515.981,Z 414.717,A 0.000,B 0.000,C 90.000,E1 345.102} C_DIS
LIN {X 0.208,Y -521.824,Z 414.704,A 0.000,B 0.000,C 90.000,E1 342.725} C_DIS
LIN {X -0.021,Y -527.877,Z 414.691,A 0.000,B 0.000,C 90.000,E1 340.423} C_DIS
LIN {X -0.091,Y -533.521,Z 414.680,A 0.000,B 0.000,C 90.000,E1 338.411} C_DIS
LIN {X -0.118,Y -539.233,Z 414.669,A 0.000,B 0.000,C 90.000,E1 336.410} C_DIS
LIN {X -0.250,Y -545.915,Z 414.656,A 0.000,B 0.000,C 90.000,E1 334.152} C_DIS
LIN {X 0.254,Y -551.077,Z 414.647,A 0.000,B 0.000,C 90.000,E1 332.410} C_DIS
LIN {X 0.120,Y -556.472,Z 414.638,A 0.000,B 0.000,C 90.000,E1 330.745} C_DIS
LIN {X 0.362,Y -560.963,Z 414.630,A 0.000,B 0.000,C 90.000,E1 329.331} C_DIS
LIN {X -0.079,Y -565.396,Z 414.622,A 0.000,B 0.000,C 90.000,E1 327.995} C_DIS
LIN {X -0.146,Y -569.825,Z 414.615,A 0.000,B 0.000,C 90.000,E1 326.628} C_DIS
LIN {X 0.000,Y -575.046,Z 414.605,A 0.000,B 0.000,C 90.000,E1 324.975} C_DIS
LIN {X 0.288,Y -581.219,Z 414.595,A 0.000,B 0.000,C 90.000,E1 323.050} C_DIS
LIN {X 0.268,Y -587.496,Z 414.584,A 0.000,B 0.000,C 90.000,E1 321.170} C_DIS
LIN {X 0.347,Y -592.102,Z 414.577,A 0.000,B 0.000,C 90.000,E1 319.828} C_DIS
LIN {X 0.289,Y -595.873,Z 414.571,A 0.000,B 0.000,C 90.000,E1 318.771} C_DIS
LIN {X -0.137,Y -603.159,Z 414.559,A 0.000,B 0.000,C 90.000,E1 316.701} C_DIS
LIN {X -0.035,Y -608.648,Z 414.551,A 0.000,B 0.000,C 90.000,E1 315.121} C_DIS
LIN {X 0.356,Y -613.233,Z 414.543,A 0.000,B 0.000,C 90.000,E1 313.785} C_DIS
LIN {X -0.035,Y -617.845,Z 414.536,A 0.000,B 0.000,C 90.000,E1 312.528} C_DIS
LIN {X -0.042,Y -623.417,Z 414.528,A 0.000,B 0.000,C 90.000,E1 310.987} C_DIS
LIN {X -0.212,Y -627.824,Z 414.521,A 0.000,B 0.000,C 90.000,E1 309.725} C_DIS
LIN {X -0.308,Y -632.077,Z 414.514,A 0.000,B 0.000,C 90.000,E1 308.463} C_DIS
LIN {X 0.163,Y -636.182,Z 414.507,A 0.000,B 0.000,C 90.000,E1 307.156} C_DIS
LIN {X -0.194,Y -640.102,Z 414.500,A 0.000,B 0.000,C 90.000,E1 305.931} C_DIS
LIN {X 0.023,Y -643.900,Z 414.493,A 0.000,B 0.000,C 90.000,E1 304.659} C_DIS
LIN {X -0.063,Y -647.585,Z 414.486,A 0.000,B 0.000,C 90.000,E1 303.420} C_DIS
LIN {X 0.112,Y -651.127,Z 414.479,A 0.000,B 0.000,C 90.000,E1 302.163} C_DIS
LIN {X 0.048,Y -653.977,Z 414.473,A 0.000,B 0.000,C 90.000,E1 301.180} C_DIS
LIN {X 0.011,Y -657.368,Z 414.466,A 0.000,B 0.000,C 90.000,E1 299.951} C_DIS
LIN {X -0.209,Y -660.531,Z 414.460,A 0.000,B 0.000,C 90.000,E1 298.743} C_DIS
LIN {X -0.127,Y -663.472,Z 414.453,A 0.000,B 0.000,C 90.000,E1 297.513} C_DIS
LIN {X 0.002,Y -666.313,Z 414.446,A 0.000,B 0.000,C 90.000,E1 296.283} C_DIS
LIN {X -0.121,Y -669.013,Z 414.439,A 0.000,B 0.000,C 90.000,E1 295.079} C_DIS
LIN {X 0.244,Y -671.019,Z 414.434,A 0.000,B 0.000,C 90.000,E1 294.079} C_DIS
LIN {X -0.074,Y -673.156,Z 414.427,A 0.000,B 0.000,C 90.000,E1 292.898} C_DIS
LIN {X 0.179,Y -674.338,Z 414.423,A 0.000,B 0.000,C 90.000,E1 292.153} C_DIS
LIN {X 0.005,Y -676.426,Z 414.414,A 0.000,B 0.000,C 90.000,E1 290.482} C_DIS
LIN {X 0.108,Y -676.920,Z 414.411,A 0.000,B 0.000,C 90.000,E1 289.993} C_DIS
LIN {X 0.263,Y -677.524,Z 414.405,A 0.000,B 0.000,C 90.000,E1 288.779} C_DIS
LIN {X 0.216,Y -677.774,Z 414.398,A 0.000,B 0.000,C 90.000,E1 287.583} C_DIS
LIN {X 0.228,Y -677.786,Z 414.393,A 0.000,B 0.000,C 90.000,E1 286.622} C_DIS
LIN {X 0.189,Y -677.505,Z 414.386,A 0.000,B 0.000,C 90.000,E1 285.426} C_DIS
LIN {X -0.035,Y -676.964,Z 414.379,A 0.000,B 0.000,C 90.000,E1 284.245} C_DIS
LIN {X 0.296,Y -675.878,Z 414.370,A 0.000,B 0.000,C 90.000,E1 282.535} C_DIS
LIN {X 0.087,Y -675.140,Z 414.364,A 0.000,B 0.000,C 90.000,E1 281.591} C_DIS
LIN {X 0.152,Y -673.817,Z 414.356,A 0.000,B 0.000,C 90.000,E1 280.141} C_DIS
LIN {X -0.285,Y -672.696,Z 414.350,A 0.000,B 0.000,C 90.000,E1 278.973} C_DIS
LIN {X -0.110,Y -671.779,Z 414.344,A 0.000,B 0.000,C 90.000,E1 277.992} C_DIS
LIN {X -0.280,Y -670.135,Z 414.335,A 0.000,B 0.000,C 90.000,E1 276.315} C_DIS
LIN {X -0.301,Y -668.885,Z 414.328,A 0.000,B 0.000,C 90.000,E1 275.106} C_DIS
LIN {X 0.320,Y -667.503,Z 414.322,A 0.000,B 0.000,C 90.000,E1 273.841} C_DIS
LIN {X 0.040,Y -665.631,Z 414.313,A 0.000,B 0.000,C 90.000,E1 272.407} C_DIS
LIN {X 0.231,Y -664.882,Z 414.309,A 0.000,B 0.000,C 90.000,E1 271.661} C_DIS
LIN {X -0.116,Y -662.853,Z 414.301,A 0.000,B 0.000,C 90.000,E1 270.229} C_DIS
LIN {X -0.287,Y -662.528,Z 414.300,A 0.000,B 0.000,C 90.000,E1 270.000} C_DIS
LIN {X 0.162,Y -660.401,Z 414.293,A 0.000,B 0.000,C 90.000,E1 268.740} C_DIS
LIN {X -0.070,Y -658.054,Z 414.286,A 0.000,B 0.000,C 90.000,E1 267.535} C_DIS
LIN {X 0.318,Y -655.364,Z 414.280,A 0.000,B 0.000,C 90.000,E1 266.274} C_DIS
LIN {X 0.207,Y -653.130,Z 414.274,A 0.000,B 0.000,C 90.000,E1 265.298} C_DIS
LIN {X -0.098,Y -649.988,Z 414.267,A 0.000,B 0.000,C 90.000,E1 264.090} C_DIS
LIN {X -0.221,Y -647.320,Z 414.262,A 0.000,B 0.000,C 90.000,E1 263.109} C_DIS
LIN {X 0.348,Y -644.455,Z 414.256,A 0.000,B 0.000,C 90.000,E1 262.064} C_DIS
LIN {X -0.319,Y -642.277,Z 414.252,A 0.000,B 0.000,C 90.000,E1 261.376} C_DIS
LIN {X 0.014,Y -638.451,Z 414.245,A 0.000,B 0.000,C 90.000,E1 260.095} C_DIS
LIN {X 0.285,Y -634.546,Z 414.238,A 0.000,B 0.000,C 90.000,E1 258.814} C_DIS
LIN {X 0.048,Y -631.340,Z 414.232,A 0.000,B 0.000,C 90.000,E1 257.825} C_DIS
LIN {X 0.115,Y -626.402,Z 414.224,A 0.000,B 0.000,C 90.000,E1 256.297} C_DIS
LIN {X 0.233,Y -621.218,Z 414.215,A 0.000,B 0.000,C 90.000,E1 254.755} C_DIS
LIN {X -0.169,Y -615.770,Z 414.207,A 0.000,B 0.000,C 90.000,E1 253.251} C_DIS
LIN {X 0.230,Y -612.047,Z 414.201,A 0.000,B 0.000,C 90.000,E1 252.181} C_DIS
LIN {X -0.085,Y -607.261,Z 414.194,A 0.000,B 0.000,C 90.000,E1 250.913} C_DIS
LIN {X 0.003,Y -601.254,Z 414.185,A 0.000,B 0.000,C 90.000,E1 249.337} C_DIS
LIN {X 0.102,Y -598.179,Z 414.181,A 0.000,B 0.000,C 90.000,E1 248.539} C_DIS
LIN {X -0.022,Y -592.879,Z 414.174,A 0.000,B 0.000,C 90.000,E1 247.230} C_DIS
LIN {X -0.229,Y -587.394,Z 414.166,A 0.000,B 0.000,C 90.000,E1 245.921} C_DIS
LIN {X 0.238,Y -581.831,Z 414.159,A 0.000,B 0.000,C 90.000,E1 244.537} C_DIS
LIN {X -0.072,Y -575.117,Z 414.150,A 0.000,B 0.000,C 90.000,E1 242.948} C_DIS
LIN {X -0.164,Y -567.376,Z 414.139,A 0.000,B 0.000,C 90.000,E1 241.051} C_DIS
LIN {X -0.153,Y -559.842,Z 414.128,A 0.000,B 0.000,C 90.000,E1 239.125} C_DIS
LIN {X -0.037,Y -552.542,Z 414.118,A 0.000,B 0.000,C 90.000,E1 237.168} C_DIS
LIN {X 0.189,Y -545.615,Z 414.107,A 0.000,B 0.000,C 90.000,E1 235.182} C_DIS
LIN {X 0.022,Y -541.700,Z 414.100,A 0.000,B 0.000,C 90.000,E1 234.069} C_DIS
LIN {X 0.127,Y -536.843,Z 414.093,A 0.000,B 0.000,C 90.000,E1 232.637} C_DIS
LIN {X 0.052,Y -530.983,Z 414.083,A 0.000,B 0.000,C 90.000,E1 230.928} C_DIS
LIN {X -0.061,Y -520.793,Z 414.065,A 0.000,B 0.000,C 90.000,E1 227.757} C_DIS
LIN {X 0.208,Y -515.531,Z 414.056,A 0.000,B 0.000,C 90.000,E1 225.972} C_DIS
LIN {X 0.085,Y -511.266,Z 414.047,A 0.000,B 0.000,C 90.000,E1 224.514} C_DIS
LIN {X -0.109,Y -504.494,Z 414.034,A 0.000,B 0.000,C 90.000,E1 222.162} C_DIS
LIN {X -0.204,Y -499.612,Z 414.024,A 0.000,B 0.000,C 90.000,E1 220.378} C_DIS
LIN {X -0.112,Y -494.017,Z 414.013,A 0.000,B 0.000,C 90.000,E1 218.257} C_DIS
LIN {X -0.148,Y -490.234,Z 414.004,A 0.000,B 0.000,C 90.000,E1 216.744} C_DIS
LIN {X 0.026,Y -484.287,Z 413.991,A 0.000,B 0.000,C 90.000,E1 214.278} C_DIS
LIN {X -0.069,Y -479.319,Z 413.979,A 0.000,B 0.000,C 90.000,E1 212.133} C_DIS
LIN {X 0.058,Y -475.032,Z 413.968,A 0.000,B 0.000,C 90.000,E1 210.256} C_DIS
LIN {X 0.089,Y -471.485,Z 413.960,A 0.000,B 0.000,C 90.000,E1 208.693} C_DIS
LIN {X 0.055,Y -467.890,Z 413.951,A 0.000,B 0.000,C 90.000,E1 207.129} C_DIS
LIN {X 0.286,Y -463.509,Z 413.940,A 0.000,B 0.000,C 90.000,E1 205.207} C_DIS
LIN {X 0.184,Y -460.470,Z 413.933,A 0.000,B 0.000,C 90.000,E1 203.951} C_DIS
LIN {X 0.181,Y -455.193,Z 413.921,A 0.000,B 0.000,C 90.000,E1 201.716} C_DIS
LIN {X -0.017,Y -450.826,Z 413.910,A 0.000,B 0.000,C 90.000,E1 199.812} C_DIS
LIN {X -0.026,Y -445.500,Z 413.896,A 0.000,B 0.000,C 90.000,E1 197.221} C_DIS
LIN {X 0.112,Y -441.901,Z 413.885,A 0.000,B 0.000,C 90.000,E1 195.245} C_DIS
LIN {X -0.066,Y -438.479,Z 413.874,A 0.000,B 0.000,C 90.000,E1 193.300} C_DIS
LIN {X 0.102,Y -435.317,Z 413.863,A 0.000,B 0.000,C 90.000,E1 191.299} C_DIS
LIN {X 0.139,Y -431.869,Z 413.850,A 0.000,B 0.000,C 90.000,E1 188.973} C_DIS
LIN {X 0.166,Y -427.997,Z 413.833,A 0.000,B 0.000,C 90.000,E1 185.967} C_DIS
LIN {X -0.073,Y -424.683,Z 413.817,A 0.000,B 0.000,C 90.000,E1 182.980} C_DIS
LIN {X -0.052,Y -422.155,Z 413.800,A 0.000,B 0.000,C 90.000,E1 179.943} C_DIS
LIN {X 0.060,Y -420.086,Z 413.775,A 0.000,B 0.000,C 90.000,E1 175.527} C_DIS
LIN {X 0.021,Y -419.724,Z 413.760,A 0.000,B 0.000,C 90.000,E1 172.818} C_DIS
LIN {X 0.166,Y -420.720,Z 413.734,A 0.000,B 0.000,C 90.000,E1 168.049} C_DIS
LIN {X -0.089,Y -422.762,Z 413.715,A 0.000,B 0.000,C 90.000,E1 164.700} C_DIS
LIN {X -0.079,Y -425.142,Z 413.700,A 0.000,B 0.000,C 90.000,E1 162.000} C_DIS
LIN {X 0.093,Y -428.501,Z 413.683,A 0.000,B 0.000,C 90.000,E1 158.954} C_DIS
LIN {X 0.108,Y -431.587,Z 413.670,A 0.000,B 0.000,C 90.000,E1 156.613} C_DIS
LIN {X 0.152,Y -435.180,Z 413.657,A 0.000,B 0.000,C 90.000,E1 154.280} C_DIS
LIN {X 0.163,Y -440.516,Z 413.641,A 0.000,B 0.000,C 90.000,E1 151.307} C_DIS
LIN {X -0.067,Y -448.057,Z 413.621,A 0.000,B 0.000,C 90.000,E1 147.740} C_DIS
LIN {X -0.145,Y -456.910,Z 413.601,A 0.000,B 0.000,C 90.000,E1 144.196} C_DIS
LIN {X -0.153,Y -465.879,Z 413.583,A 0.000,B 0.000,C 90.000,E1 141.009} C_DIS
LIN {X 0.037,Y -471.681,Z 413.573,A 0.000,B 0.000,C 90.000,E1 139.094} C_DIS
LIN {X 0.073,Y -475.497,Z 413.566,A 0.000,B 0.000,C 90.000,E1 137.838} C_DIS
LIN {X -0.153,Y -479.117,Z 413.559,A 0.000,B 0.000,C 90.000,E1 136.620} C_DIS
LIN {X 0.205,Y -481.738,Z 413.554,A 0.000,B 0.000,C 90.000,E1 135.648} C_DIS
LIN {X -0.085,Y -484.136,Z 413.549,A 0.000,B 0.000,C 90.000,E1 134.757} C_DIS
LIN {X -0.205,Y -487.136,Z 413.542,A 0.000,B 0.000,C 90.000,E1 133.542} C_DIS
LIN {X -0.087,Y -489.111,Z 413.537,A 0.000,B 0.000,C 90.000,E1 132.609} C_DIS
LIN {X -0.110,Y -491.352,Z 413.530,A 0.000,B 0.000,C 90.000,E1 131.391} C_DIS
LIN {X 0.057,Y -492.618,Z 413.525,A 0.000,B 0.000,C 90.000,E1 130.458} C_DIS
LIN {X 0.066,Y -493.277,Z 413.521,A 0.000,B 0.000,C 90.000,E1 129.850} C_DIS
LIN {X -0.071,Y -493.985,Z 413.516,A 0.000,B 0.000,C 90.000,E1 128.955} C_DIS
LIN {X 0.186,Y -494.116,Z 413.511,A 0.000,B 0.000,C 90.000,E1 128.016} C_DIS
LIN {X -0.246,Y -493.585,Z 413.506,A 0.000,B 0.000,C 90.000,E1 127.156} C_DIS
LIN {X 0.007,Y -492.646,Z 413.501,A 0.000,B 0.000,C 90.000,E1 126.217} C_DIS
LIN {X -0.043,Y -491.260,Z 413.496,A 0.000,B 0.000,C 90.000,E1 125.311} C_DIS
LIN {X 0.054,Y -490.266,Z 413.493,A 0.000,B 0.000,C 90.000,E1 124.692} C_DIS
LIN {X 0.143,Y -488.987,Z 413.489,A 0.000,B 0.000,C 90.000,E1 124.072} C_DIS
LIN {X 0.056,Y -486.660,Z 413.484,A 0.000,B 0.000,C 90.000,E1 123.166} C_DIS
LIN {X 0.118,Y -484.890,Z 413.481,A 0.000,B 0.000,C 90.000,E1 122.546} C_DIS
LIN {X -0.279,Y -481.893,Z 413.476,A 0.000,B 0.000,C 90.000,E1 121.671} C_DIS
LIN {X 0.155,Y -479.779,Z 413.472,A 0.000,B 0.000,C 90.000,E1 121.003} C_DIS
LIN {X -0.101,Y -474.963,Z 413.466,A 0.000,B 0.000,C 90.000,E1 119.795} C_DIS
LIN {X -0.021,Y -470.430,Z 413.459,A 0.000,B 0.000,C 90.000,E1 118.693} C_DIS
LIN {X 0.000,Y -465.713,Z 413.453,A 0.000,B 0.000,C 90.000,E1 117.590} C_DIS
LIN {X 0.121,Y -460.044,Z 413.446,A 0.000,B 0.000,C 90.000,E1 116.309} C_DIS
LIN {X -0.108,Y -453.454,Z 413.438,A 0.000,B 0.000,C 90.000,E1 114.899} C_DIS
LIN {X -0.134,Y -447.599,Z 413.431,A 0.000,B 0.000,C 90.000,E1 113.643} C_DIS
LIN {X -0.174,Y -447.582,Z 413.431,A 0.000,B 0.000,C 90.000,E1 113.643} C_DIS
LIN {X -0.044,Y -457.066,Z 413.410,A 0.000,B 0.000,C 90.000,E1 109.885} C_DIS
LIN {X -0.078,Y -460.128,Z 413.402,A 0.000,B 0.000,C 90.000,E1 108.290} C_DIS
LIN {X -0.239,Y -467.259,Z 413.384,A 0.000,B 0.000,C 90.000,E1 105.134} C_DIS
LIN {X 0.137,Y -467.956,Z 413.382,A 0.000,B 0.000,C 90.000,E1 104.773} C_DIS
LIN {X 0.101,Y -476.176,Z 413.356,A 0.000,B 0.000,C 90.000,E1 100.074} C_DIS
LIN {X -0.123,Y -482.082,Z 413.330,A 0.000,B 0.000,C 90.000,E1 95.448} C_DIS
LIN {X 0.107,Y -485.502,Z 413.305,A 0.000,B 0.000,C 90.000,E1 90.802} C_DIS
LIN {X 0.140,Y -486.384,Z 413.281,A 0.000,B 0.000,C 90.000,E1 86.502} C_DIS
LIN {X -0.036,Y -486.361,Z 413.279,A 0.000,B 0.000,C 90.000,E1 86.216} C_DIS
LIN {X 0.048,Y -484.686,Z 413.253,A 0.000,B 0.000,C 90.000,E1 81.602} C_DIS
LIN {X -0.053,Y -480.609,Z 413.228,A 0.000,B 0.000,C 90.000,E1 76.992} C_DIS
LIN {X -0.195,Y -480.251,Z 413.226,A 0.000,B 0.000,C 90.000,E1 76.700} C_DIS
LIN {X 0.161,Y -474.080,Z 413.200,A 0.000,B 0.000,C 90.000,E1 72.000} C_DIS
LIN {X -0.057,Y -468.207,Z 413.182,A 0.000,B 0.000,C 90.000,E1 68.827} C_DIS
LIN {X -0.097,Y -468.242,Z 413.182,A 0.000,B 0.000,C 90.000,E1 68.827} C_DIS
LIN {X -0.240,Y -474.804,Z 413.178,A 0.000,B 0.000,C 90.000,E1 67.975} C_DIS
LIN {X -0.123,Y -486.775,Z 413.169,A 0.000,B 0.000,C 90.000,E1 66.410} C_DIS
LIN {X -0.060,Y -493.664,Z 413.164,A 0.000,B 0.000,C 90.000,E1 65.485} C_DIS
LIN {X -0.166,Y -500.196,Z 413.159,A 0.000,B 0.000,C 90.000,E1 64.588} C_DIS
LIN {X -0.039,Y -504.296,Z 413.155,A 0.000,B 0.000,C 90.000,E1 63.973} C_DIS
LIN {X 0.157,Y -509.071,Z 413.151,A 0.000,B 0.000,C 90.000,E1 63.204} C_DIS
LIN {X -0.056,Y -513.605,Z 413.147,A 0.000,B 0.000,C 90.000,E1 62.487} C_DIS
LIN {X -0.057,Y -516.889,Z 413.144,A 0.000,B 0.000,C 90.000,E1 61.897} C_DIS
LIN {X -0.197,Y -520.628,Z 413.140,A 0.000,B 0.000,C 90.000,E1 61.179} C_DIS
LIN {X 0.149,Y -523.873,Z 413.136,A 0.000,B 0.000,C 90.000,E1 60.411} C_DIS
LIN {X -0.234,Y -526.248,Z 413.133,A 0.000,B 0.000,C 90.000,E1 59.871} C_DIS
LIN {X -0.144,Y -528.313,Z 413.129,A 0.000,B 0.000,C 90.000,E1 59.282} C_DIS
LIN {X -0.076,Y -530.973,Z 413.124,A 0.000,B 0.000,C 90.000,E1 58.408} C_DIS
LIN {X 0.326,Y -532.385,Z 413.121,A 0.000,B 0.000,C 90.000,E1 57.788} C_DIS
LIN {X -0.006,Y -534.026,Z 413.116,A 0.000,B 0.000,C 90.000,E1 56.962} C_DIS
LIN {X 0.124,Y -535.134,Z 413.112,A 0.000,B 0.000,C 90.000,E1 56.087} C_DIS
LIN {X 0.122,Y -535.661,Z 413.109,A 0.000,B 0.000,C 90.000,E1 55.515} C_DIS
LIN {X -0.178,Y -535.942,Z 413.104,A 0.000,B 0.000,C 90.000,E1 54.689} C_DIS
LIN {X -0.164,Y -535.958,Z 413.099,A 0.000,B 0.000,C 90.000,E1 53.829} C_DIS
LIN {X -0.147,Y -535.683,Z 413.094,A 0.000,B 0.000,C 90.000,E1 52.970} C_DIS
LIN {X -0.133,Y -535.089,Z 413.089,A 0.000,B 0.000,C 90.000,E1 52.110} C_DIS
LIN {X 0.201,Y -533.704,Z 413.082,A 0.000,B 0.000,C 90.000,E1 50.642} C_DIS
LIN {X -0.237,Y -532.492,Z 413.075,A 0.000,B 0.000,C 90.000,E1 49.542} C_DIS
LIN {X 0.065,Y -531.382,Z 413.070,A 0.000,B 0.000,C 90.000,E1 48.647} C_DIS
LIN {X -0.134,Y -529.276,Z 413.062,A 0.000,B 0.000,C 90.000,E1 47.229} C_DIS
LIN {X 0.277,Y -526.333,Z 413.051,A 0.000,B 0.000,C 90.000,E1 45.162} C_DIS
LIN {X -0.129,Y -523.662,Z 413.040,A 0.000,B 0.000,C 90.000,E1 43.176} C_DIS
LIN {X -0.163,Y -521.539,Z 413.030,A 0.000,B 0.000,C 90.000,E1 41.434} C_DIS
LIN {X 0.185,Y -519.452,Z 413.020,A 0.000,B 0.000,C 90.000,E1 39.644} C_DIS
LIN {X 0.225,Y -517.737,Z 413.012,A 0.000,B 0.000,C 90.000,E1 38.177} C_DIS
LIN {X -0.147,Y -515.630,Z 413.003,A 0.000,B 0.000,C 90.000,E1 36.457} C_DIS
LIN {X -0.146,Y -513.374,Z 412.993,A 0.000,B 0.000,C 90.000,E1 34.692} C_DIS
LIN {X -0.039,Y -511.823,Z 412.986,A 0.000,B 0.000,C 90.000,E1 33.499} C_DIS
LIN {X -0.242,Y -510.159,Z 412.980,A 0.000,B 0.000,C 90.000,E1 32.339} C_DIS
LIN {X 0.294,Y -508.251,Z 412.971,A 0.000,B 0.000,C 90.000,E1 30.797} C_DIS
LIN {X 0.043,Y -505.474,Z 412.960,A 0.000,B 0.000,C 90.000,E1 28.743} C_DIS
LIN {X 0.064,Y -503.229,Z 412.950,A 0.000,B 0.000,C 90.000,E1 26.950} C_DIS
LIN {X -0.062,Y -500.583,Z 412.936,A 0.000,B 0.000,C 90.000,E1 24.567} C_DIS
LIN {X 0.019,Y -498.223,Z 412.923,A 0.000,B 0.000,C 90.000,E1 22.153} C_DIS
LIN {X -0.033,Y -495.934,Z 412.906,A 0.000,B 0.000,C 90.000,E1 19.141} C_DIS
LIN {X -0.105,Y -494.910,Z 412.898,A 0.000,B 0.000,C 90.000,E1 17.638} C_DIS
LIN {X 0.173,Y -493.625,Z 412.888,A 0.000,B 0.000,C 90.000,E1 15.788} C_DIS
LIN {X -0.167,Y -492.350,Z 412.876,A 0.000,B 0.000,C 90.000,E1 13.703} C_DIS
LIN {X 0.177,Y -491.319,Z 412.864,A 0.000,B 0.000,C 90.000,E1 11.535} C_DIS
LIN {X -0.084,Y -490.695,Z 412.852,A 0.000,B 0.000,C 90.000,E1 9.434} C_DIS
LIN {X -0.033,Y -490.470,Z 412.841,A 0.000,B 0.000,C 90.000,E1 7.296} C_DIS
LIN {X 0.165,Y -490.322,Z 412.837,A 0.000,B 0.000,C 90.000,E1 6.663} C_DIS
LIN {X 0.080,Y -490.538,Z 412.830,A 0.000,B 0.000,C 90.000,E1 5.454} C_DIS
LIN {X -0.207,Y -491.742,Z 412.810,A 0.000,B 0.000,C 90.000,E1 1.833} C_DIS
LIN {X 0.170,Y -495.265,Z 412.787,A 0.000,B 0.000,C 90.000,E1 357.650} C_DIS
LIN {X -0.124,Y -497.498,Z 412.777,A 0.000,B 0.000,C 90.000,E1 355.869} C_DIS
LIN {X 0.034,Y -500.456,Z 412.765,A 0.000,B 0.000,C 90.000,E1 353.742} C_DIS
LIN {X -0.114,Y -503.811,Z 412.754,A 0.000,B 0.000,C 90.000,E1 351.659} C_DIS
LIN {X 0.190,Y -510.579,Z 412.734,A 0.000,B 0.000,C 90.000,E1 348.049} C_DIS
LIN {X 0.152,Y -517.344,Z 412.717,A 0.000,B 0.000,C 90.000,E1 345.102} C_DIS
LIN {X -0.023,Y -523.935,Z 412.703,A 0.000,B 0.000,C 90.000,E1 342.489} C_DIS
LIN {X -0.198,Y -530.055,Z 412.690,A 0.000,B 0.000,C 90.000,E1 340.188} C_DIS
LIN {X -0.230,Y -534.900,Z 412.680,A 0.000,B 0.000,C 90.000,E1 338.465} C_DIS
LIN {X -0.208,Y -541.444,Z 412.668,A 0.000,B 0.000,C 90.000,E1 336.177} C_DIS
LIN {X -0.298,Y -549.017,Z 412.653,A 0.000,B 0.000,C 90.000,E1 333.640} C_DIS
LIN {X 0.051,Y -555.117,Z 412.643,A 0.000,B 0.000,C 90.000,E1 331.641} C_DIS
LIN {X -0.070,Y -558.760,Z 412.636,A 0.000,B 0.000,C 90.000,E1 330.539} C_DIS
LIN {X 0.133,Y -562.365,Z 412.630,A 0.000,B 0.000,C 90.000,E1 329.410} C_DIS
LIN {X 0.010,Y -566.816,Z 412.623,A 0.000,B 0.000,C 90.000,E1 328.043} C_DIS
LIN {X -0.211,Y -572.105,Z 412.613,A 0.000,B 0.000,C 90.000,E1 326.421} C_DIS
LIN {X -0.166,Y -576.493,Z 412.606,A 0.000,B 0.000,C 90.000,E1 325.055} C_DIS
LIN {X 0.151,Y -582.700,Z 412.595,A 0.000,B 0.000,C 90.000,E1 323.130} C_DIS
LIN {X 0.163,Y -588.984,Z 412.585,A 0.000,B 0.000,C 90.000,E1 321.251} C_DIS
LIN {X 0.266,Y -593.660,Z 412.577,A 0.000,B 0.000,C 90.000,E1 319.908} C_DIS
LIN {X 0.000,Y -598.270,Z 412.570,A 0.000,B 0.000,C 90.000,E1 318.609} C_DIS
LIN {X -0.188,Y -602.870,Z 412.563,A 0.000,B 0.000,C 90.000,E1 317.310} C_DIS
LIN {X 0.300,Y -606.541,Z 412.557,A 0.000,B 0.000,C 90.000,E1 316.215} C_DIS
LIN {X 0.225,Y -611.090,Z 412.550,A 0.000,B 0.000,C 90.000,E1 314.919} C_DIS
LIN {X 0.394,Y -614.798,Z 412.544,A 0.000,B 0.000,C 90.000,E1 313.866} C_DIS
LIN {X 0.030,Y -619.439,Z 412.537,A 0.000,B 0.000,C 90.000,E1 312.609} C_DIS
LIN {X 0.058,Y -624.988,Z 412.528,A 0.000,B 0.000,C 90.000,E1 311.067} C_DIS
LIN {X 0.050,Y -628.571,Z 412.523,A 0.000,B 0.000,C 90.000,E1 310.048} C_DIS
LIN {X 0.010,Y -632.046,Z 412.517,A 0.000,B 0.000,C 90.000,E1 309.036} C_DIS
LIN {X -0.415,Y -636.202,Z 412.510,A 0.000,B 0.000,C 90.000,E1 307.810} C_DIS
LIN {X 0.125,Y -640.226,Z 412.503,A 0.000,B 0.000,C 90.000,E1 306.503} C_DIS
LIN {X 0.351,Y -644.057,Z 412.496,A 0.000,B 0.000,C 90.000,E1 305.231} C_DIS
LIN {X 0.274,Y -647.839,Z 412.489,A 0.000,B 0.000,C 90.000,E1 303.992} C_DIS
LIN {X 0.262,Y -651.447,Z 412.482,A 0.000,B 0.000,C 90.000,E1 302.752} C_DIS
LIN {X 0.399,Y -655.723,Z 412.474,A 0.000,B 0.000,C 90.000,E1 301.258} C_DIS
LIN {X 0.276,Y -659.774,Z 412.466,A 0.000,B 0.000,C 90.000,E1 299.795} C_DIS
LIN {X -0.234,Y -662.948,Z 412.459,A 0.000,B 0.000,C 90.000,E1 298.615} C_DIS
LIN {X -0.257,Y -665.286,Z 412.453,A 0.000,B 0.000,C 90.000,E1 297.641} C_DIS
LIN {X -0.099,Y -668.070,Z 412.447,A 0.000,B 0.000,C 90.000,E1 296.411} C_DIS
LIN {X 0.247,Y -670.239,Z 412.441,A 0.000,B 0.000,C 90.000,E1 295.412} C_DIS
LIN {X 0.366,Y -673.247,Z 412.433,A 0.000,B 0.000,C 90.000,E1 293.951} C_DIS
LIN {X -0.003,Y -674.479,Z 412.429,A 0.000,B 0.000,C 90.000,E1 293.259} C_DIS
LIN {X 0.177,Y -676.061,Z 412.424,A 0.000,B 0.000,C 90.000,E1 292.280} C_DIS
LIN {X 0.044,Y -677.832,Z 412.415,A 0.000,B 0.000,C 90.000,E1 290.610} C_DIS
LIN {X 0.158,Y -678.276,Z 412.412,A 0.000,B 0.000,C 90.000,E1 290.120} C_DIS
LIN {X 0.340,Y -678.826,Z 412.405,A 0.000,B 0.000,C 90.000,E1 288.906} C_DIS
LIN {X -0.330,Y -679.040,Z 412.399,A 0.000,B 0.000,C 90.000,E1 287.764} C_DIS
LIN {X -0.149,Y -678.947,Z 412.392,A 0.000,B 0.000,C 90.000,E1 286.551} C_DIS
LIN {X -0.359,Y -678.510,Z 412.385,A 0.000,B 0.000,C 90.000,E1 285.371} C_DIS
LIN {X 0.303,Y -677.933,Z 412.380,A 0.000,B 0.000,C 90.000,E1 284.356} C_DIS
LIN {X 0.080,Y -676.964,Z 412.373,A 0.000,B 0.000,C 90.000,E1 283.175} C_DIS
LIN {X -0.015,Y -676.602,Z 412.371,A 0.000,B 0.000,C 90.000,E1 282.703} C_DIS
LIN {X 0.305,Y -675.747,Z 412.365,A 0.000,B 0.000,C 90.000,E1 281.715} C_DIS
LIN {X 0.269,Y -673.738,Z 412.355,A 0.000,B 0.000,C 90.000,E1 279.792} C_DIS
LIN {X 0.247,Y -672.034,Z 412.345,A 0.000,B 0.000,C 90.000,E1 278.106} C_DIS
LIN {X 0.166,Y -670.573,Z 412.337,A 0.000,B 0.000,C 90.000,E1 276.663} C_DIS
LIN {X 0.157,Y -669.424,Z 412.330,A 0.000,B 0.000,C 90.000,E1 275.454} C_DIS
LIN {X 0.014,Y -667.921,Z 412.322,A 0.000,B 0.000,C 90.000,E1 274.012} C_DIS
LIN {X 0.067,Y -666.845,Z 412.317,A 0.000,B 0.000,C 90.000,E1 273.037} C_DIS
LIN {X -0.084,Y -665.546,Z 412.310,A 0.000,B 0.000,C 90.000,E1 271.835} C_DIS
LIN {X -0.062,Y -664.471,Z 412.305,A 0.000,B 0.000,C 90.000,E1 270.859} C_DIS
LIN {X -0.070,Y -663.219,Z 412.299,A 0.000,B 0.000,C 90.000,E1 269.885} C_DIS
LIN {X -0.271,Y -661.238,Z 412.293,A 0.000,B 0.000,C 90.000,E1 268.682} C_DIS
LIN {X 0.171,Y -658.970,Z 412.286,A 0.000,B 0.000,C 90.000,E1 267.421} C_DIS
LIN {X -0.279,Y -655.840,Z 412.278,A 0.000,B 0.000,C 90.000,E1 265.988} C_DIS
LIN {X -0.181,Y -654.179,Z 412.274,A 0.000,B 0.000,C 90.000,E1 265.241} C_DIS
LIN {X 0.179,Y -651.100,Z 412.267,A 0.000,B 0.000,C 90.000,E1 263.976} C_DIS
LIN {X -0.086,Y -647.769,Z 412.260,A 0.000,B 0.000,C 90.000,E1 262.761} C_DIS
LIN {X 0.242,Y -644.201,Z 412.253,A 0.000,B 0.000,C 90.000,E1 261.489} C_DIS
LIN {X 0.139,Y -641.199,Z 412.247,A 0.000,B 0.000,C 90.000,E1 260.500} C_DIS
LIN {X 0.168,Y -636.587,Z 412.239,A 0.000,B 0.000,C 90.000,E1 258.993} C_DIS
LIN {X -0.093,Y -632.619,Z 412.232,A 0.000,B 0.000,C 90.000,E1 257.757} C_DIS
LIN {X 0.015,Y -627.726,Z 412.224,A 0.000,B 0.000,C 90.000,E1 256.228} C_DIS
LIN {X 0.220,Y -623.433,Z 412.216,A 0.000,B 0.000,C 90.000,E1 254.936} C_DIS
LIN {X -0.144,Y -617.984,Z 412.208,A 0.000,B 0.000,C 90.000,E1 253.433} C_DIS
LIN {X 0.286,Y -614.288,Z 412.202,A 0.000,B 0.000,C 90.000,E1 252.362} C_DIS
LIN {X 0.008,Y -609.514,Z 412.195,A 0.000,B 0.000,C 90.000,E1 251.094} C_DIS
LIN {X -0.145,Y -604.531,Z 412.188,A 0.000,B 0.000,C 90.000,E1 249.806} C_DIS
LIN {X 0.266,Y -600.464,Z 412.182,A 0.000,B 0.000,C 90.000,E1 248.720} C_DIS
LIN {X 0.181,Y -595.186,Z 412.175,A 0.000,B 0.000,C 90.000,E1 247.411} C_DIS
LIN {X 0.014,Y -589.717,Z 412.167,A 0.000,B 0.000,C 90.000,E1 246.102} C_DIS
LIN {X -0.252,Y -584.158,Z 412.160,A 0.000,B 0.000,C 90.000,E1 244.793} C_DIS
LIN {X 0.266,Y -577.458,Z 412.151,A 0.000,B 0.000,C 90.000,E1 243.127} C_DIS
LIN {X -0.039,Y -569.659,Z 412.140,A 0.000,B 0.000,C 90.000,E1 241.257} C_DIS
LIN {X 0.021,Y -562.103,Z 412.130,A 0.000,B 0.000,C 90.000,E1 239.331} C_DIS
LIN {X 0.189,Y -554.780,Z 412.119,A 0.000,B 0.000,C 90.000,E1 237.375} C_DIS
LIN {X -0.243,Y -546.852,Z 412.106,A 0.000,B 0.000,C 90.000,E1 235.182} C_DIS
LIN {X -0.038,Y -541.957,Z 412.099,A 0.000,B 0.000,C 90.000,E1 233.749} C_DIS
LIN {X -0.259,Y -538.114,Z 412.092,A 0.000,B 0.000,C 90.000,E1 232.637} C_DIS
LIN {X 0.110,Y -532.264,Z 412.083,A 0.000,B 0.000,C 90.000,E1 230.884} C_DIS
LIN {X 0.079,Y -522.959,Z 412.067,A 0.000,B 0.000,C 90.000,E1 228.000} C_DIS
LIN {X 0.019,Y -517.702,Z 412.057,A 0.000,B 0.000,C 90.000,E1 226.257} C_DIS
LIN {X -0.154,Y -512.530,Z 412.047,A 0.000,B 0.000,C 90.000,E1 224.514} C_DIS
LIN {X 0.029,Y -505.754,Z 412.034,A 0.000,B 0.000,C 90.000,E1 222.123} C_DIS
LIN {X 0.007,Y -500.853,Z 412.024,A 0.000,B 0.000,C 90.000,E1 220.334} C_DIS
LIN {X -0.080,Y -494.503,Z 412.011,A 0.000,B 0.000,C 90.000,E1 217.935} C_DIS
LIN {X 0.127,Y -489.943,Z 412.001,A 0.000,B 0.000,C 90.000,E1 216.091} C_DIS
LIN {X -0.220,Y -484.782,Z 411.989,A 0.000,B 0.000,C 90.000,E1 213.992} C_DIS
LIN {X 0.101,Y -479.833,Z 411.977,A 0.000,B 0.000,C 90.000,E1 211.799} C_DIS
LIN {X -0.221,Y -474.820,Z 411.965,A 0.000,B 0.000,C 90.000,E1 209.667} C_DIS
LIN {X -0.190,Y -471.267,Z 411.956,A 0.000,B 0.000,C 90.000,E1 208.103} C_DIS
LIN {X 0.186,Y -467.631,Z 411.947,A 0.000,B 0.000,C 90.000,E1 206.488} C_DIS
LIN {X -0.208,Y -463.191,Z 411.937,A 0.000,B 0.000,C 90.000,E1 204.643} C_DIS
LIN {X -0.049,Y -458.566,Z 411.926,A 0.000,B 0.000,C 90.000,E1 202.717} C_DIS
LIN {X 0.003,Y -454.134,Z 411.916,A 0.000,B 0.000,C 90.000,E1 200.791} C_DIS
LIN {X 0.111,Y -447.859,Z 411.899,A 0.000,B 0.000,C 90.000,E1 197.873} C_DIS
LIN {X 0.028,Y -443.535,Z 411.887,A 0.000,B 0.000,C 90.000,E1 195.607} C_DIS
LIN {X -0.003,Y -440.075,Z 411.876,A 0.000,B 0.000,C 90.000,E1 193.647} C_DIS
LIN {X -0.178,Y -436.310,Z 411.863,A 0.000,B 0.000,C 90.000,E1 191.366} C_DIS
LIN {X -0.028,Y -432.845,Z 411.850,A 0.000,B 0.000,C 90.000,E1 189.029} C_DIS
LIN {X -0.015,Y -428.912,Z 411.834,A 0.000,B 0.000,C 90.000,E1 186.030} C_DIS
LIN {X -0.178,Y -425.568,Z 411.817,A 0.000,B 0.000,C 90.000,E1 183.037} C_DIS
LIN {X -0.125,Y -423.006,Z 411.800,A 0.000,B 0.000,C 90.000,E1 180.000} C_DIS
LIN {X 0.032,Y -420.902,Z 411.776,A 0.000,B 0.000,C 90.000,E1 175.584} C_DIS
LIN {X 0.021,Y -420.544,Z 411.760,A 0.000,B 0.000,C 90.000,E1 172.875} C_DIS
LIN {X 0.129,Y -421.497,Z 411.734,A 0.000,B 0.000,C 90.000,E1 168.117} C_DIS
LIN {X -0.072,Y -423.270,Z 411.717,A 0.000,B 0.000,C 90.000,E1 165.102} C_DIS
LIN {X 0.037,Y -425.890,Z 411.700,A 0.000,B 0.000,C 90.000,E1 162.054} C_DIS
LIN {X -0.113,Y -428.836,Z 411.685,A 0.000,B 0.000,C 90.000,E1 159.390} C_DIS
LIN {X -0.093,Y -431.901,Z 411.672,A 0.000,B 0.000,C 90.000,E1 157.050} C_DIS
LIN {X 0.188,Y -436.520,Z 411.656,A 0.000,B 0.000,C 90.000,E1 154.024} C_DIS
LIN {X 0.078,Y -442.575,Z 411.638,A 0.000,B 0.000,C 90.000,E1 150.745} C_DIS
LIN {X -0.065,Y -449.626,Z 411.619,A 0.000,B 0.000,C 90.000,E1 147.502} C_DIS
LIN {X -0.319,Y -458.671,Z 411.600,A 0.000,B 0.000,C 90.000,E1 143.989} C_DIS
LIN {X -0.022,Y -466.876,Z 411.584,A 0.000,B 0.000,C 90.000,E1 141.090} C_DIS
LIN {X -0.166,Y -472.744,Z 411.573,A 0.000,B 0.000,C 90.000,E1 139.218} C_DIS
LIN {X -0.075,Y -476.601,Z 411.566,A 0.000,B 0.000,C 90.000,E1 137.957} C_DIS
LIN {X 0.035,Y -480.267,Z 411.560,A 0.000,B 0.000,C 90.000,E1 136.701} C_DIS
LIN {X -0.275,Y -482.885,Z 411.554,A 0.000,B 0.000,C 90.000,E1 135.810} C_DIS
LIN {X 0.132,Y -485.390,Z 411.549,A 0.000,B 0.000,C 90.000,E1 134.838} C_DIS
LIN {X 0.185,Y -489.125,Z 411.541,A 0.000,B 0.000,C 90.000,E1 133.299} C_DIS
LIN {X -0.003,Y -491.085,Z 411.536,A 0.000,B 0.000,C 90.000,E1 132.405} C_DIS
LIN {X -0.037,Y -493.305,Z 411.529,A 0.000,B 0.000,C 90.000,E1 131.191} C_DIS
LIN {X 0.056,Y -494.880,Z 411.522,A 0.000,B 0.000,C 90.000,E1 129.967} C_DIS
LIN {X -0.057,Y -495.656,Z 411.517,A 0.000,B 0.000,C 90.000,E1 129.072} C_DIS
LIN {X -0.164,Y -495.874,Z 411.512,A 0.000,B 0.000,C 90.000,E1 128.177} C_DIS
LIN {X 0.003,Y -495.892,Z 411.510,A 0.000,B 0.000,C 90.000,E1 127.855} C_DIS
LIN {X -0.018,Y -495.253,Z 411.505,A 0.000,B 0.000,C 90.000,E1 126.950} C_DIS
LIN {X 0.255,Y -494.232,Z 411.500,A 0.000,B 0.000,C 90.000,E1 126.011} C_DIS
LIN {X 0.225,Y -492.852,Z 411.495,A 0.000,B 0.000,C 90.000,E1 125.105} C_DIS
LIN {X -0.072,Y -491.811,Z 411.492,A 0.000,B 0.000,C 90.000,E1 124.532} C_DIS
LIN {X 0.027,Y -490.449,Z 411.488,A 0.000,B 0.000,C 90.000,E1 123.913} C_DIS
LIN {X -0.048,Y -488.141,Z 411.483,A 0.000,B 0.000,C 90.000,E1 123.007} C_DIS
LIN {X -0.239,Y -486.315,Z 411.480,A 0.000,B 0.000,C 90.000,E1 122.418} C_DIS
LIN {X 0.049,Y -483.255,Z 411.475,A 0.000,B 0.000,C 90.000,E1 121.465} C_DIS
LIN {X -0.168,Y -481.109,Z 411.471,A 0.000,B 0.000,C 90.000,E1 120.875} C_DIS
LIN {X -0.176,Y -476.873,Z 411.465,A 0.000,B 0.000,C 90.000,E1 119.795} C_DIS
LIN {X -0.077,Y -471.669,Z 411.459,A 0.000,B 0.000,C 90.000,E1 118.537} C_DIS
LIN {X -0.022,Y -467.584,Z 411.453,A 0.000,B 0.000,C 90.000,E1 117.590} C_DIS
LIN {X 0.127,Y -461.843,Z 411.446,A 0.000,B 0.000,C 90.000,E1 116.309} C_DIS
LIN {X 0.087,Y -454.474,Z 411.437,A 0.000,B 0.000,C 90.000,E1 114.719} C_DIS
LIN {X -0.086,Y -448.150,Z 411.430,A 0.000,B 0.000,C 90.000,E1 113.387} C_DIS
LIN {X -0.125,Y -448.142,Z 411.430,A 0.000,B 0.000,C 90.000,E1 113.387} C_DIS
LIN {X -0.234,Y -457.418,Z 411.410,A 0.000,B 0.000,C 90.000,E1 109.758} C_DIS
LIN {X -0.151,Y -466.065,Z 411.387,A 0.000,B 0.000,C 90.000,E1 105.607} C_DIS
LIN {X 0.023,Y -467.634,Z 411.383,A 0.000,B 0.000,C 90.000,E1 104.954} C_DIS
LIN {X -0.054,Y -469.561,Z 411.376,A 0.000,B 0.000,C 90.000,E1 103.703} C_DIS
LIN {X -0.019,Y -475.855,Z 411.357,A 0.000,B 0.000,C 90.000,E1 100.254} C_DIS
LIN {X -0.181,Y -476.329,Z 411.355,A 0.000,B 0.000,C 90.000,E1 99.962} C_DIS
LIN {X -0.234,Y -481.830,Z 411.331,A 0.000,B 0.000,C 90.000,E1 95.625} C_DIS
LIN {X 0.092,Y -482.181,Z 411.329,A 0.000,B 0.000,C 90.000,E1 95.277} C_DIS
LIN {X 0.027,Y -485.335,Z 411.305,A 0.000,B 0.000,C 90.000,E1 90.974} C_DIS
LIN {X -0.149,Y -485.534,Z 411.304,A 0.000,B 0.000,C 90.000,E1 90.688} C_DIS
LIN {X 0.058,Y -486.332,Z 411.282,A 0.000,B 0.000,C 90.000,E1 86.674} C_DIS
LIN {X 0.192,Y -486.287,Z 411.278,A 0.000,B 0.000,C 90.000,E1 86.045} C_DIS
LIN {X -0.088,Y -484.694,Z 411.254,A 0.000,B 0.000,C 90.000,E1 81.781} C_DIS
LIN {X -0.219,Y -484.569,Z 411.253,A 0.000,B 0.000,C 90.000,E1 81.489} C_DIS
LIN {X 0.129,Y -480.507,Z 411.227,A 0.000,B 0.000,C 90.000,E1 76.825} C_DIS
LIN {X 0.026,Y -474.260,Z 411.201,A 0.000,B 0.000,C 90.000,E1 72.181} C_DIS
LIN {X -0.007,Y -473.794,Z 411.199,A 0.000,B 0.000,C 90.000,E1 71.873} C_DIS
LIN {X 0.095,Y -468.561,Z 411.184,A 0.000,B 0.000,C 90.000,E1 69.028} C_DIS
LIN {X 0.055,Y -468.574,Z 411.184,A 0.000,B 0.000,C 90.000,E1 69.028} C_DIS
LIN {X -0.150,Y -476.721,Z 411.178,A 0.000,B 0.000,C 90.000,E1 67.975} C_DIS
LIN {X 0.064,Y -487.425,Z 411.170,A 0.000,B 0.000,C 90.000,E1 66.561} C_DIS
LIN {X -0.117,Y -494.304,Z 411.165,A 0.000,B 0.000,C 90.000,E1 65.665} C_DIS
LIN {X 0.045,Y -501.869,Z 411.159,A 0.000,B 0.000,C 90.000,E1 64.588} C_DIS
LIN {X -0.268,Y -505.914,Z 411.156,A 0.000,B 0.000,C 90.000,E1 64.024} C_DIS
LIN {X 0.125,Y -509.713,Z 411.152,A 0.000,B 0.000,C 90.000,E1 63.384} C_DIS
LIN {X 0.096,Y -513.300,Z 411.149,A 0.000,B 0.000,C 90.000,E1 62.794} C_DIS
LIN {X -0.137,Y -516.718,Z 411.146,A 0.000,B 0.000,C 90.000,E1 62.231} C_DIS
LIN {X -0.115,Y -519.762,Z 411.142,A 0.000,B 0.000,C 90.000,E1 61.641} C_DIS
LIN {X 0.094,Y -521.960,Z 411.140,A 0.000,B 0.000,C 90.000,E1 61.179} C_DIS
LIN {X 0.158,Y -524.517,Z 411.137,A 0.000,B 0.000,C 90.000,E1 60.589} C_DIS
LIN {X -0.076,Y -527.961,Z 411.132,A 0.000,B 0.000,C 90.000,E1 59.744} C_DIS
LIN {X 0.024,Y -529.975,Z 411.129,A 0.000,B 0.000,C 90.000,E1 59.154} C_DIS
LIN {X -0.040,Y -531.712,Z 411.125,A 0.000,B 0.000,C 90.000,E1 58.584} C_DIS
LIN {X 0.072,Y -533.813,Z 411.121,A 0.000,B 0.000,C 90.000,E1 57.709} C_DIS
LIN {X 0.212,Y -534.896,Z 411.118,A 0.000,B 0.000,C 90.000,E1 57.120} C_DIS
LIN {X -0.097,Y -536.109,Z 411.113,A 0.000,B 0.000,C 90.000,E1 56.294} C_DIS
LIN {X -0.088,Y -536.860,Z 411.108,A 0.000,B 0.000,C 90.000,E1 55.435} C_DIS
LIN {X 0.065,Y -537.093,Z 411.103,A 0.000,B 0.000,C 90.000,E1 54.562} C_DIS
LIN {X 0.089,Y -537.083,Z 411.098,A 0.000,B 0.000,C 90.000,E1 53.703} C_DIS
LIN {X 0.115,Y -536.766,Z 411.094,A 0.000,B 0.000,C 90.000,E1 52.844} C_DIS
LIN {X 0.141,Y -535.899,Z 411.087,A 0.000,B 0.000,C 90.000,E1 51.698} C_DIS
LIN {X 0.071,Y -534.773,Z 411.081,A 0.000,B 0.000,C 90.000,E1 50.561} C_DIS
LIN {X -0.013,Y -533.144,Z 411.073,A 0.000,B 0.000,C 90.000,E1 49.138} C_DIS
LIN {X -0.114,Y -531.511,Z 411.067,A 0.000,B 0.000,C 90.000,E1 48.000} C_DIS
LIN {X 0.083,Y -529.363,Z 411.059,A 0.000,B 0.000,C 90.000,E1 46.539} C_DIS
LIN {X 0.115,Y -526.476,Z 411.047,A 0.000,B 0.000,C 90.000,E1 44.514} C_DIS
LIN {X -0.162,Y -524.588,Z 411.039,A 0.000,B 0.000,C 90.000,E1 43.095} C_DIS
LIN {X 0.263,Y -522.818,Z 411.031,A 0.000,B 0.000,C 90.000,E1 41.595} C_DIS
LIN {X -0.091,Y -520.704,Z 411.022,A 0.000,B 0.000,C 90.000,E1 39.886} C_DIS
LIN {X 0.300,Y -518.996,Z 411.013,A 0.000,B 0.000,C 90.000,E1 38.382} C_DIS
LIN {X -0.048,Y -516.863,Z 411.004,A 0.000,B 0.000,C 90.000,E1 36.664} C_DIS
LIN {X -0.022,Y -514.635,Z 410.994,A 0.000,B 0.000,C 90.000,E1 34.898} C_DIS
LIN {X 0.103,Y -513.089,Z 410.987,A 0.000,B 0.000,C 90.000,E1 33.706} C_DIS
LIN {X 0.261,Y -511.038,Z 410.979,A 0.000,B 0.000,C 90.000,E1 32.212} C_DIS
LIN {X 0.117,Y -509.122,Z 410.971,A 0.000,B 0.000,C 90.000,E1 30.747} C_DIS
LIN {X -0.103,Y -506.363,Z 410.959,A 0.000,B 0.000,C 90.000,E1 28.693} C_DIS
LIN {X -0.132,Y -504.504,Z 410.951,A 0.000,B 0.000,C 90.000,E1 27.206} C_DIS
LIN {X -0.142,Y -501.506,Z 410.936,A 0.000,B 0.000,C 90.000,E1 24.515} C_DIS
LIN {X 0.163,Y -499.159,Z 410.923,A 0.000,B 0.000,C 90.000,E1 22.078} C_DIS
LIN {X -0.032,Y -496.867,Z 410.906,A 0.000,B 0.000,C 90.000,E1 19.087} C_DIS
LIN {X -0.084,Y -495.851,Z 410.898,A 0.000,B 0.000,C 90.000,E1 17.583} C_DIS
LIN {X -0.255,Y -494.595,Z 410.888,A 0.000,B 0.000,C 90.000,E1 15.788} C_DIS
LIN {X -0.189,Y -493.164,Z 410.874,A 0.000,B 0.000,C 90.000,E1 13.355} C_DIS
LIN {X -0.120,Y -491.974,Z 410.857,A 0.000,B 0.000,C 90.000,E1 10.310} C_DIS
LIN {X 0.135,Y -491.566,Z 410.840,A 0.000,B 0.000,C 90.000,E1 7.239} C_DIS
LIN {X 0.230,Y -491.531,Z 410.835,A 0.000,B 0.000,C 90.000,E1 6.315} C_DIS
LIN {X 0.211,Y -491.891,Z 410.823,A 0.000,B 0.000,C 90.000,E1 4.188} C_DIS
LIN {X -0.205,Y -493.995,Z 410.802,A 0.000,B 0.000,C 90.000,E1 0.286} C_DIS
LIN {X -0.075,Y -497.191,Z 410.784,A 0.000,B 0.000,C 90.000,E1 357.078} C_DIS
LIN {X -0.066,Y -500.423,Z 410.770,A 0.000,B 0.000,C 90.000,E1 354.666} C_DIS
LIN {X 0.075,Y -504.595,Z 410.755,A 0.000,B 0.000,C 90.000,E1 351.951} C_DIS
LIN {X -0.123,Y -511.915,Z 410.734,A 0.000,B 0.000,C 90.000,E1 348.105} C_DIS
LIN {X -0.122,Y -519.445,Z 410.716,A 0.000,B 0.000,C 90.000,E1 344.866} C_DIS
LIN {X -0.234,Y -525.374,Z 410.703,A 0.000,B 0.000,C 90.000,E1 342.543} C_DIS
LIN {X -0.048,Y -530.696,Z 410.692,A 0.000,B 0.000,C 90.000,E1 340.496} C_DIS
LIN {X 0.139,Y -536.316,Z 410.680,A 0.000,B 0.000,C 90.000,E1 338.465} C_DIS
LIN {X 0.208,Y -542.870,Z 410.668,A 0.000,B 0.000,C 90.000,E1 336.177} C_DIS
LIN {X 0.169,Y -550.421,Z 410.654,A 0.000,B 0.000,C 90.000,E1 333.640} C_DIS
LIN {X 0.071,Y -556.564,Z 410.643,A 0.000,B 0.000,C 90.000,E1 331.691} C_DIS
LIN {X -0.234,Y -561.062,Z 410.635,A 0.000,B 0.000,C 90.000,E1 330.333} C_DIS
LIN {X -0.194,Y -565.595,Z 410.627,A 0.000,B 0.000,C 90.000,E1 328.948} C_DIS
LIN {X -0.263,Y -570.033,Z 410.620,A 0.000,B 0.000,C 90.000,E1 327.582} C_DIS
LIN {X -0.287,Y -576.211,Z 410.609,A 0.000,B 0.000,C 90.000,E1 325.674} C_DIS
LIN {X -0.146,Y -583.274,Z 410.597,A 0.000,B 0.000,C 90.000,E1 323.497} C_DIS
LIN {X -0.323,Y -588.658,Z 410.588,A 0.000,B 0.000,C 90.000,E1 321.904} C_DIS
LIN {X 0.200,Y -595.198,Z 410.578,A 0.000,B 0.000,C 90.000,E1 319.989} C_DIS
LIN {X -0.042,Y -599.840,Z 410.571,A 0.000,B 0.000,C 90.000,E1 318.690} C_DIS
LIN {X 0.000,Y -603.523,Z 410.565,A 0.000,B 0.000,C 90.000,E1 317.634} C_DIS
LIN {X 0.306,Y -608.116,Z 410.557,A 0.000,B 0.000,C 90.000,E1 316.296} C_DIS
LIN {X 0.257,Y -612.662,Z 410.550,A 0.000,B 0.000,C 90.000,E1 315.000} C_DIS
LIN {X -0.422,Y -616.361,Z 410.544,A 0.000,B 0.000,C 90.000,E1 314.028} C_DIS
LIN {X -0.039,Y -621.952,Z 410.536,A 0.000,B 0.000,C 90.000,E1 312.447} C_DIS
LIN {X 0.037,Y -627.491,Z 410.527,A 0.000,B 0.000,C 90.000,E1 310.906} C_DIS
LIN {X -0.193,Y -632.860,Z 410.519,A 0.000,B 0.000,C 90.000,E1 309.402} C_DIS
LIN {X -0.222,Y -637.849,Z 410.510,A 0.000,B 0.000,C 90.000,E1 307.890} C_DIS
LIN {X 0.351,Y -641.890,Z 410.503,A 0.000,B 0.000,C 90.000,E1 306.583} C_DIS
LIN {X -0.291,Y -645.735,Z 410.497,A 0.000,B 0.000,C 90.000,E1 305.391} C_DIS
LIN {X 0.027,Y -649.552,Z 410.490,A 0.000,B 0.000,C 90.000,E1 304.119} C_DIS
LIN {X 0.126,Y -653.859,Z 410.481,A 0.000,B 0.000,C 90.000,E1 302.625} C_DIS
LIN {X 0.314,Y -658.135,Z 410.473,A 0.000,B 0.000,C 90.000,E1 301.131} C_DIS
LIN {X 0.239,Y -662.181,Z 410.465,A 0.000,B 0.000,C 90.000,E1 299.667} C_DIS
LIN {X -0.232,Y -665.299,Z 410.458,A 0.000,B 0.000,C 90.000,E1 298.487} C_DIS
LIN {X -0.224,Y -667.655,Z 410.453,A 0.000,B 0.000,C 90.000,E1 297.513} C_DIS
LIN {X 0.011,Y -671.465,Z 410.443,A 0.000,B 0.000,C 90.000,E1 295.796} C_DIS
LIN {X 0.088,Y -673.466,Z 410.438,A 0.000,B 0.000,C 90.000,E1 294.823} C_DIS
LIN {X -0.378,Y -675.476,Z 410.433,A 0.000,B 0.000,C 90.000,E1 293.898} C_DIS
LIN {X 0.262,Y -677.424,Z 410.426,A 0.000,B 0.000,C 90.000,E1 292.642} C_DIS
LIN {X 0.038,Y -678.628,Z 410.419,A 0.000,B 0.000,C 90.000,E1 291.461} C_DIS
LIN {X 0.219,Y -679.615,Z 410.413,A 0.000,B 0.000,C 90.000,E1 290.248} C_DIS
LIN {X -0.345,Y -679.908,Z 410.409,A 0.000,B 0.000,C 90.000,E1 289.577} C_DIS
LIN {X -0.264,Y -680.024,Z 410.405,A 0.000,B 0.000,C 90.000,E1 288.852} C_DIS
LIN {X -0.013,Y -680.066,Z 410.399,A 0.000,B 0.000,C 90.000,E1 287.873} C_DIS
LIN {X -0.019,Y -679.786,Z 410.393,A 0.000,B 0.000,C 90.000,E1 286.677} C_DIS
LIN {X -0.071,Y -679.150,Z 410.385,A 0.000,B 0.000,C 90.000,E1 285.245} C_DIS
LIN {X -0.230,Y -678.530,Z 410.379,A 0.000,B 0.000,C 90.000,E1 284.300} C_DIS
LIN {X 0.220,Y -677.539,Z 410.373,A 0.000,B 0.000,C 90.000,E1 283.063} C_DIS
LIN {X -0.014,Y -676.352,Z 410.366,A 0.000,B 0.000,C 90.000,E1 281.883} C_DIS
LIN {X -0.110,Y -673.862,Z 410.354,A 0.000,B 0.000,C 90.000,E1 279.726} C_DIS
LIN {X 0.179,Y -671.571,Z 410.342,A 0.000,B 0.000,C 90.000,E1 277.530} C_DIS
LIN {X -0.163,Y -669.715,Z 410.331,A 0.000,B 0.000,C 90.000,E1 275.625} C_DIS
LIN {X -0.351,Y -668.285,Z 410.323,A 0.000,B 0.000,C 90.000,E1 274.188} C_DIS
LIN {X 0.095,Y -666.837,Z 410.315,A 0.000,B 0.000,C 90.000,E1 272.694} C_DIS
LIN {X -0.195,Y -665.496,Z 410.307,A 0.000,B 0.000,C 90.000,E1 271.260} C_DIS
LIN {X 0.141,Y -664.956,Z 410.304,A 0.000,B 0.000,C 90.000,E1 270.745} C_DIS
LIN {X 0.140,Y -663.726,Z 410.299,A 0.000,B 0.000,C 90.000,E1 269.771} C_DIS
LIN {X 0.120,Y -662.171,Z 410.293,A 0.000,B 0.000,C 90.000,E1 268.797} C_DIS
LIN {X -0.083,Y -660.026,Z 410.287,A 0.000,B 0.000,C 90.000,E1 267.593} C_DIS
LIN {X 0.059,Y -658.687,Z 410.283,A 0.000,B 0.000,C 90.000,E1 266.846} C_DIS
LIN {X -0.195,Y -656.204,Z 410.276,A 0.000,B 0.000,C 90.000,E1 265.641} C_DIS
LIN {X -0.089,Y -654.537,Z 410.272,A 0.000,B 0.000,C 90.000,E1 264.894} C_DIS
LIN {X -0.149,Y -652.148,Z 410.266,A 0.000,B 0.000,C 90.000,E1 263.913} C_DIS
LIN {X 0.178,Y -648.848,Z 410.259,A 0.000,B 0.000,C 90.000,E1 262.648} C_DIS
LIN {X -0.117,Y -645.386,Z 410.252,A 0.000,B 0.000,C 90.000,E1 261.432} C_DIS
LIN {X 0.269,Y -641.636,Z 410.245,A 0.000,B 0.000,C 90.000,E1 260.151} C_DIS
LIN {X -0.324,Y -637.047,Z 410.237,A 0.000,B 0.000,C 90.000,E1 258.701} C_DIS
LIN {X 0.225,Y -633.889,Z 410.232,A 0.000,B 0.000,C 90.000,E1 257.645} C_DIS
LIN {X -0.073,Y -629.865,Z 410.225,A 0.000,B 0.000,C 90.000,E1 256.408} C_DIS
LIN {X 0.167,Y -625.613,Z 410.217,A 0.000,B 0.000,C 90.000,E1 255.117} C_DIS
LIN {X -0.159,Y -620.195,Z 410.209,A 0.000,B 0.000,C 90.000,E1 253.614} C_DIS
LIN {X 0.304,Y -616.493,Z 410.203,A 0.000,B 0.000,C 90.000,E1 252.543} C_DIS
LIN {X 0.061,Y -611.738,Z 410.196,A 0.000,B 0.000,C 90.000,E1 251.275} C_DIS
LIN {X 0.006,Y -607.789,Z 410.190,A 0.000,B 0.000,C 90.000,E1 250.242} C_DIS
LIN {X -0.172,Y -602.742,Z 410.183,A 0.000,B 0.000,C 90.000,E1 248.954} C_DIS
LIN {X -0.129,Y -598.521,Z 410.177,A 0.000,B 0.000,C 90.000,E1 247.901} C_DIS
LIN {X 0.076,Y -593.103,Z 410.170,A 0.000,B 0.000,C 90.000,E1 246.561} C_DIS
LIN {X 0.104,Y -587.591,Z 410.162,A 0.000,B 0.000,C 90.000,E1 245.229} C_DIS
LIN {X -0.213,Y -579.765,Z 410.152,A 0.000,B 0.000,C 90.000,E1 243.384} C_DIS
LIN {X -0.144,Y -574.174,Z 410.145,A 0.000,B 0.000,C 90.000,E1 242.025} C_DIS
LIN {X -0.247,Y -566.514,Z 410.134,A 0.000,B 0.000,C 90.000,E1 240.127} C_DIS
LIN {X -0.176,Y -558.067,Z 410.122,A 0.000,B 0.000,C 90.000,E1 237.916} C_DIS
LIN {X 0.003,Y -549.055,Z 410.108,A 0.000,B 0.000,C 90.000,E1 235.388} C_DIS
LIN {X -0.072,Y -544.193,Z 410.100,A 0.000,B 0.000,C 90.000,E1 233.989} C_DIS
LIN {X 0.082,Y -539.389,Z 410.092,A 0.000,B 0.000,C 90.000,E1 232.557} C_DIS
LIN {X -0.274,Y -534.510,Z 410.084,A 0.000,B 0.000,C 90.000,E1 231.170} C_DIS
LIN {X 0.353,Y -528.770,Z 410.075,A 0.000,B 0.000,C 90.000,E1 229.380} C_DIS
LIN {X -0.047,Y -521.611,Z 410.062,A 0.000,B 0.000,C 90.000,E1 227.106} C_DIS
LIN {X 0.215,Y -516.354,Z 410.052,A 0.000,B 0.000,C 90.000,E1 225.324} C_DIS
LIN {X 0.107,Y -512.080,Z 410.044,A 0.000,B 0.000,C 90.000,E1 223.866} C_DIS
LIN {X 0.180,Y -507.001,Z 410.034,A 0.000,B 0.000,C 90.000,E1 222.081} C_DIS
LIN {X 0.136,Y -502.088,Z 410.024,A 0.000,B 0.000,C 90.000,E1 220.297} C_DIS
LIN {X 0.154,Y -495.751,Z 410.011,A 0.000,B 0.000,C 90.000,E1 217.890} C_DIS
LIN {X 0.147,Y -491.946,Z 410.002,A 0.000,B 0.000,C 90.000,E1 216.377} C_DIS
LIN {X -0.147,Y -486.740,Z 409.990,A 0.000,B 0.000,C 90.000,E1 214.278} C_DIS
LIN {X -0.177,Y -481.745,Z 409.978,A 0.000,B 0.000,C 90.000,E1 212.133} C_DIS
LIN {X 0.008,Y -477.448,Z 409.968,A 0.000,B 0.000,C 90.000,E1 210.256} C_DIS
LIN {X 0.085,Y -473.919,Z 409.960,A 0.000,B 0.000,C 90.000,E1 208.693} C_DIS
LIN {X -0.071,Y -471.032,Z 409.953,A 0.000,B 0.000,C 90.000,E1 207.462} C_DIS
LIN {X 0.151,Y -468.112,Z 409.946,A 0.000,B 0.000,C 90.000,E1 206.181} C_DIS
LIN {X -0.164,Y -464.367,Z 409.937,A 0.000,B 0.000,C 90.000,E1 204.643} C_DIS
LIN {X 0.100,Y -460.532,Z 409.928,A 0.000,B 0.000,C 90.000,E1 203.025} C_DIS
LIN {X 0.102,Y -455.291,Z 409.916,A 0.000,B 0.000,C 90.000,E1 200.791} C_DIS
LIN {X -0.056,Y -449.658,Z 409.901,A 0.000,B 0.000,C 90.000,E1 198.236} C_DIS
LIN {X 0.194,Y -444.631,Z 409.887,A 0.000,B 0.000,C 90.000,E1 195.607} C_DIS
LIN {X 0.189,Y -441.164,Z 409.876,A 0.000,B 0.000,C 90.000,E1 193.647} C_DIS
LIN {X 0.041,Y -437.366,Z 409.863,A 0.000,B 0.000,C 90.000,E1 191.366} C_DIS
LIN {X -0.150,Y -433.385,Z 409.849,A 0.000,B 0.000,C 90.000,E1 188.746} C_DIS
LIN {X -0.056,Y -429.456,Z 409.832,A 0.000,B 0.000,C 90.000,E1 185.739} C_DIS
LIN {X 0.133,Y -426.533,Z 409.817,A 0.000,B 0.000,C 90.000,E1 183.037} C_DIS
LIN {X -0.156,Y -423.697,Z 409.798,A 0.000,B 0.000,C 90.000,E1 179.714} C_DIS
LIN {X 0.033,Y -421.695,Z 409.774,A 0.000,B 0.000,C 90.000,E1 175.298} C_DIS
LIN {X 0.019,Y -421.364,Z 409.761,A 0.000,B 0.000,C 90.000,E1 172.932} C_DIS
LIN {X -0.046,Y -421.887,Z 409.740,A 0.000,B 0.000,C 90.000,E1 169.218} C_DIS
LIN {X -0.009,Y -423.402,Z 409.723,A 0.000,B 0.000,C 90.000,E1 166.172} C_DIS
LIN {X -0.169,Y -426.354,Z 409.703,A 0.000,B 0.000,C 90.000,E1 162.489} C_DIS
LIN {X 0.233,Y -429.217,Z 409.688,A 0.000,B 0.000,C 90.000,E1 159.752} C_DIS
LIN {X 0.089,Y -432.710,Z 409.673,A 0.000,B 0.000,C 90.000,E1 157.102} C_DIS
LIN {X 0.238,Y -437.882,Z 409.654,A 0.000,B 0.000,C 90.000,E1 153.768} C_DIS
LIN {X 0.013,Y -444.028,Z 409.636,A 0.000,B 0.000,C 90.000,E1 150.511} C_DIS
LIN {X 0.011,Y -450.486,Z 409.620,A 0.000,B 0.000,C 90.000,E1 147.582} C_DIS
LIN {X 0.058,Y -459.567,Z 409.600,A 0.000,B 0.000,C 90.000,E1 144.036} C_DIS
LIN {X 0.066,Y -466.929,Z 409.586,A 0.000,B 0.000,C 90.000,E1 141.492} C_DIS
LIN {X -0.005,Y -473.805,Z 409.574,A 0.000,B 0.000,C 90.000,E1 139.299} C_DIS
LIN {X -0.252,Y -477.685,Z 409.567,A 0.000,B 0.000,C 90.000,E1 138.081} C_DIS
LIN {X -0.121,Y -481.405,Z 409.560,A 0.000,B 0.000,C 90.000,E1 136.824} C_DIS
LIN {X -0.067,Y -484.056,Z 409.555,A 0.000,B 0.000,C 90.000,E1 135.891} C_DIS
LIN {X 0.012,Y -486.639,Z 409.550,A 0.000,B 0.000,C 90.000,E1 134.960} C_DIS
LIN {X 0.276,Y -489.667,Z 409.543,A 0.000,B 0.000,C 90.000,E1 133.704} C_DIS
LIN {X -0.268,Y -491.750,Z 409.538,A 0.000,B 0.000,C 90.000,E1 132.852} C_DIS
LIN {X 0.066,Y -493.052,Z 409.535,A 0.000,B 0.000,C 90.000,E1 132.204} C_DIS
LIN {X -0.075,Y -494.723,Z 409.530,A 0.000,B 0.000,C 90.000,E1 131.310} C_DIS
LIN {X -0.047,Y -495.618,Z 409.526,A 0.000,B 0.000,C 90.000,E1 130.701} C_DIS
LIN {X -0.154,Y -496.715,Z 409.521,A 0.000,B 0.000,C 90.000,E1 129.806} C_DIS
LIN {X -0.249,Y -497.418,Z 409.516,A 0.000,B 0.000,C 90.000,E1 128.910} C_DIS
LIN {X 0.054,Y -497.599,Z 409.511,A 0.000,B 0.000,C 90.000,E1 127.971} C_DIS
LIN {X -0.077,Y -497.524,Z 409.509,A 0.000,B 0.000,C 90.000,E1 127.684} C_DIS
LIN {X -0.170,Y -496.909,Z 409.504,A 0.000,B 0.000,C 90.000,E1 126.790} C_DIS
LIN {X -0.172,Y -495.817,Z 409.499,A 0.000,B 0.000,C 90.000,E1 125.884} C_DIS
LIN {X 0.244,Y -494.942,Z 409.496,A 0.000,B 0.000,C 90.000,E1 125.231} C_DIS
LIN {X 0.222,Y -493.338,Z 409.491,A 0.000,B 0.000,C 90.000,E1 124.326} C_DIS
LIN {X -0.092,Y -491.158,Z 409.486,A 0.000,B 0.000,C 90.000,E1 123.452} C_DIS
LIN {X 0.006,Y -489.591,Z 409.482,A 0.000,B 0.000,C 90.000,E1 122.832} C_DIS
LIN {X 0.091,Y -487.746,Z 409.479,A 0.000,B 0.000,C 90.000,E1 122.212} C_DIS
LIN {X -0.275,Y -484.636,Z 409.474,A 0.000,B 0.000,C 90.000,E1 121.337} C_DIS
LIN {X 0.182,Y -482.447,Z 409.471,A 0.000,B 0.000,C 90.000,E1 120.669} C_DIS
LIN {X -0.019,Y -479.436,Z 409.466,A 0.000,B 0.000,C 90.000,E1 119.922} C_DIS
LIN {X -0.114,Y -473.574,Z 409.459,A 0.000,B 0.000,C 90.000,E1 118.537} C_DIS
LIN {X 0.195,Y -470.159,Z 409.454,A 0.000,B 0.000,C 90.000,E1 117.719} C_DIS
LIN {X -0.033,Y -464.393,Z 409.447,A 0.000,B 0.000,C 90.000,E1 116.488} C_DIS
LIN {X 0.134,Y -456.279,Z 409.437,A 0.000,B 0.000,C 90.000,E1 114.719} C_DIS
LIN {X -0.025,Y -448.714,Z 409.429,A 0.000,B 0.000,C 90.000,E1 113.131} C_DIS
LIN {X -0.064,Y -448.710,Z 409.428,A 0.000,B 0.000,C 90.000,E1 113.131} C_DIS
LIN {X 0.118,Y -457.008,Z 409.411,A 0.000,B 0.000,C 90.000,E1 109.885} C_DIS
LIN {X -0.073,Y -458.260,Z 409.407,A 0.000,B 0.000,C 90.000,E1 109.268} C_DIS
LIN {X 0.124,Y -466.424,Z 409.386,A 0.000,B 0.000,C 90.000,E1 105.426} C_DIS
LIN {X -0.152,Y -467.929,Z 409.382,A 0.000,B 0.000,C 90.000,E1 104.828} C_DIS
LIN {X -0.038,Y -475.506,Z 409.358,A 0.000,B 0.000,C 90.000,E1 100.423} C_DIS
LIN {X 0.182,Y -476.145,Z 409.356,A 0.000,B 0.000,C 90.000,E1 100.084} C_DIS
LIN {X -0.003,Y -482.058,Z 409.330,A 0.000,B 0.000,C 90.000,E1 95.454} C_DIS
LIN {X -0.214,Y -485.486,Z 409.305,A 0.000,B 0.000,C 90.000,E1 90.859} C_DIS
LIN {X -0.181,Y -486.386,Z 409.281,A 0.000,B 0.000,C 90.000,E1 86.560} C_DIS
LIN {X 0.129,Y -486.363,Z 409.279,A 0.000,B 0.000,C 90.000,E1 86.216} C_DIS
LIN {X 0.212,Y -484.689,Z 409.254,A 0.000,B 0.000,C 90.000,E1 81.602} C_DIS
LIN {X -0.172,Y -482.721,Z 409.243,A 0.000,B 0.000,C 90.000,E1 79.803} C_DIS
LIN {X 0.111,Y -480.619,Z 409.228,A 0.000,B 0.000,C 90.000,E1 76.992} C_DIS
LIN {X -0.031,Y -480.284,Z 409.226,A 0.000,B 0.000,C 90.000,E1 76.700} C_DIS
LIN {X -0.126,Y -474.108,Z 409.200,A 0.000,B 0.000,C 90.000,E1 72.054} C_DIS
LIN {X -0.047,Y -468.917,Z 409.185,A 0.000,B 0.000,C 90.000,E1 69.263} C_DIS
LIN {X -0.087,Y -468.933,Z 409.185,A 0.000,B 0.000,C 90.000,E1 69.263} C_DIS
LIN {X -0.041,Y -478.657,Z 409.178,A 0.000,B 0.000,C 90.000,E1 67.975} C_DIS
LIN {X -0.274,Y -489.313,Z 409.170,A 0.000,B 0.000,C 90.000,E1 66.613} C_DIS
LIN {X 0.018,Y -496.076,Z 409.165,A 0.000,B 0.000,C 90.000,E1 65.665} C_DIS
LIN {X -0.272,Y -502.561,Z 409.160,A 0.000,B 0.000,C 90.000,E1 64.793} C_DIS
LIN {X -0.097,Y -507.571,Z 409.156,A 0.000,B 0.000,C 90.000,E1 64.024} C_DIS
LIN {X -0.146,Y -511.339,Z 409.152,A 0.000,B 0.000,C 90.000,E1 63.435} C_DIS
LIN {X -0.221,Y -514.028,Z 409.150,A 0.000,B 0.000,C 90.000,E1 62.999} C_DIS
LIN {X 0.083,Y -518.164,Z 409.146,A 0.000,B 0.000,C 90.000,E1 62.231} C_DIS
LIN {X 0.118,Y -521.153,Z 409.143,A 0.000,B 0.000,C 90.000,E1 61.641} C_DIS
LIN {X 0.337,Y -523.296,Z 409.140,A 0.000,B 0.000,C 90.000,E1 61.179} C_DIS
LIN {X 0.255,Y -526.388,Z 409.136,A 0.000,B 0.000,C 90.000,E1 60.461} C_DIS
LIN {X -0.108,Y -528.666,Z 409.133,A 0.000,B 0.000,C 90.000,E1 59.921} C_DIS
LIN {X 0.001,Y -530.716,Z 409.130,A 0.000,B 0.000,C 90.000,E1 59.331} C_DIS
LIN {X 0.100,Y -533.226,Z 409.125,A 0.000,B 0.000,C 90.000,E1 58.456} C_DIS
LIN {X 0.239,Y -534.673,Z 409.122,A 0.000,B 0.000,C 90.000,E1 57.867} C_DIS
LIN {X -0.072,Y -536.230,Z 409.117,A 0.000,B 0.000,C 90.000,E1 57.041} C_DIS
LIN {X -0.367,Y -537.055,Z 409.114,A 0.000,B 0.000,C 90.000,E1 56.501} C_DIS
LIN {X 0.094,Y -537.888,Z 409.109,A 0.000,B 0.000,C 90.000,E1 55.595} C_DIS
LIN {X -0.185,Y -538.251,Z 409.104,A 0.000,B 0.000,C 90.000,E1 54.769} C_DIS
LIN {X -0.147,Y -538.298,Z 409.099,A 0.000,B 0.000,C 90.000,E1 53.909} C_DIS
LIN {X -0.107,Y -538.016,Z 409.095,A 0.000,B 0.000,C 90.000,E1 53.050} C_DIS
LIN {X -0.058,Y -537.217,Z 409.088,A 0.000,B 0.000,C 90.000,E1 51.904} C_DIS
LIN {X 0.308,Y -536.127,Z 409.082,A 0.000,B 0.000,C 90.000,E1 50.723} C_DIS
LIN {X 0.244,Y -534.470,Z 409.074,A 0.000,B 0.000,C 90.000,E1 49.299} C_DIS
LIN {X -0.182,Y -533.294,Z 409.069,A 0.000,B 0.000,C 90.000,E1 48.485} C_DIS
LIN {X 0.045,Y -531.190,Z 409.061,A 0.000,B 0.000,C 90.000,E1 47.025} C_DIS
LIN {X 0.120,Y -528.224,Z 409.050,A 0.000,B 0.000,C 90.000,E1 45.000} C_DIS
LIN {X -0.193,Y -525.886,Z 409.040,A 0.000,B 0.000,C 90.000,E1 43.299} C_DIS
LIN {X -0.099,Y -524.098,Z 409.032,A 0.000,B 0.000,C 90.000,E1 41.838} C_DIS
LIN {X -0.085,Y -521.957,Z 409.023,A 0.000,B 0.000,C 90.000,E1 40.092} C_DIS
LIN {X 0.002,Y -520.256,Z 409.015,A 0.000,B 0.000,C 90.000,E1 38.624} C_DIS
LIN {X 0.057,Y -518.465,Z 409.007,A 0.000,B 0.000,C 90.000,E1 37.156} C_DIS
LIN {X -0.241,Y -516.625,Z 408.998,A 0.000,B 0.000,C 90.000,E1 35.724} C_DIS
LIN {X 0.267,Y -514.758,Z 408.990,A 0.000,B 0.000,C 90.000,E1 34.199} C_DIS
LIN {X -0.056,Y -512.362,Z 408.980,A 0.000,B 0.000,C 90.000,E1 32.467} C_DIS
LIN {X 0.158,Y -509.987,Z 408.971,A 0.000,B 0.000,C 90.000,E1 30.669} C_DIS
LIN {X -0.047,Y -507.252,Z 408.959,A 0.000,B 0.000,C 90.000,E1 28.615} C_DIS
LIN {X -0.128,Y -504.717,Z 408.947,A 0.000,B 0.000,C 90.000,E1 26.539} C_DIS
LIN {X 0.020,Y -502.101,Z 408.934,A 0.000,B 0.000,C 90.000,E1 24.131} C_DIS
LIN {X 0.149,Y -499.850,Z 408.921,A 0.000,B 0.000,C 90.000,E1 21.716} C_DIS
LIN {X -0.014,Y -497.613,Z 408.904,A 0.000,B 0.000,C 90.000,E1 18.725} C_DIS
LIN {X -0.052,Y -496.587,Z 408.896,A 0.000,B 0.000,C 90.000,E1 17.221} C_DIS
LIN {X -0.212,Y -495.362,Z 408.886,A 0.000,B 0.000,C 90.000,E1 15.426} C_DIS
LIN {X -0.149,Y -494.155,Z 408.874,A 0.000,B 0.000,C 90.000,E1 13.300} C_DIS
LIN {X 0.062,Y -493.084,Z 408.859,A 0.000,B 0.000,C 90.000,E1 10.546} C_DIS
LIN {X -0.227,Y -492.650,Z 408.840,A 0.000,B 0.000,C 90.000,E1 7.239} C_DIS
LIN {X 0.045,Y -492.969,Z 408.825,A 0.000,B 0.000,C 90.000,E1 4.473} C_DIS
LIN {X 0.168,Y -495.005,Z 408.803,A 0.000,B 0.000,C 90.000,E1 0.516} C_DIS
LIN {X -0.140,Y -498.806,Z 408.782,A 0.000,B 0.000,C 90.000,E1 356.788} C_DIS
LIN {X -0.202,Y -502.543,Z 408.767,A 0.000,B 0.000,C 90.000,E1 354.090} C_DIS
LIN {X -0.097,Y -507.957,Z 408.749,A 0.000,B 0.000,C 90.000,E1 350.792} C_DIS
LIN {X 0.011,Y -514.510,Z 408.731,A 0.000,B 0.000,C 90.000,E1 347.521} C_DIS
LIN {X 0.021,Y -518.643,Z 408.721,A 0.000,B 0.000,C 90.000,E1 345.755} C_DIS
LIN {X 0.117,Y -521.559,Z 408.714,A 0.000,B 0.000,C 90.000,E1 344.574} C_DIS
LIN {X 0.055,Y -526.786,Z 408.703,A 0.000,B 0.000,C 90.000,E1 342.543} C_DIS
LIN {X -0.220,Y -532.125,Z 408.692,A 0.000,B 0.000,C 90.000,E1 340.550} C_DIS
LIN {X -0.188,Y -537.733,Z 408.681,A 0.000,B 0.000,C 90.000,E1 338.539} C_DIS
LIN {X -0.131,Y -545.115,Z 408.667,A 0.000,B 0.000,C 90.000,E1 335.973} C_DIS
LIN {X -0.102,Y -551.825,Z 408.654,A 0.000,B 0.000,C 90.000,E1 333.717} C_DIS
LIN {X -0.176,Y -558.011,Z 408.643,A 0.000,B 0.000,C 90.000,E1 331.769} C_DIS
LIN {X 0.184,Y -564.282,Z 408.632,A 0.000,B 0.000,C 90.000,E1 329.793} C_DIS
LIN {X -0.198,Y -568.798,Z 408.625,A 0.000,B 0.000,C 90.000,E1 328.456} C_DIS
LIN {X 0.150,Y -572.343,Z 408.619,A 0.000,B 0.000,C 90.000,E1 327.327} C_DIS
LIN {X -0.126,Y -577.666,Z 408.610,A 0.000,B 0.000,C 90.000,E1 325.722} C_DIS
LIN {X -0.110,Y -583.834,Z 408.599,A 0.000,B 0.000,C 90.000,E1 323.829} C_DIS
LIN {X 0.005,Y -588.358,Z 408.592,A 0.000,B 0.000,C 90.000,E1 322.477} C_DIS
LIN {X -0.090,Y -595.780,Z 408.580,A 0.000,B 0.000,C 90.000,E1 320.356} C_DIS
LIN {X 0.130,Y -600.455,Z 408.572,A 0.000,B 0.000,C 90.000,E1 319.013} C_DIS
LIN {X -0.270,Y -604.228,Z 408.567,A 0.000,B 0.000,C 90.000,E1 318.000} C_DIS
LIN {X 0.123,Y -610.583,Z 408.556,A 0.000,B 0.000,C 90.000,E1 316.134} C_DIS
LIN {X -0.050,Y -616.075,Z 408.548,A 0.000,B 0.000,C 90.000,E1 314.595} C_DIS
LIN {X 0.188,Y -622.590,Z 408.538,A 0.000,B 0.000,C 90.000,E1 312.771} C_DIS
LIN {X -0.053,Y -627.200,Z 408.531,A 0.000,B 0.000,C 90.000,E1 311.515} C_DIS
LIN {X -0.037,Y -630.899,Z 408.525,A 0.000,B 0.000,C 90.000,E1 310.496} C_DIS
LIN {X -0.042,Y -634.497,Z 408.519,A 0.000,B 0.000,C 90.000,E1 309.483} C_DIS
LIN {X -0.034,Y -639.490,Z 408.511,A 0.000,B 0.000,C 90.000,E1 307.971} C_DIS
LIN {X 0.055,Y -643.557,Z 408.504,A 0.000,B 0.000,C 90.000,E1 306.710} C_DIS
LIN {X -0.040,Y -647.414,Z 408.497,A 0.000,B 0.000,C 90.000,E1 305.471} C_DIS
LIN {X 0.312,Y -651.248,Z 408.490,A 0.000,B 0.000,C 90.000,E1 304.199} C_DIS
LIN {X -0.003,Y -656.276,Z 408.481,A 0.000,B 0.000,C 90.000,E1 302.498} C_DIS
LIN {X 0.236,Y -660.507,Z 408.472,A 0.000,B 0.000,C 90.000,E1 301.003} C_DIS
LIN {X 0.210,Y -664.571,Z 408.464,A 0.000,B 0.000,C 90.000,E1 299.539} C_DIS
LIN {X -0.223,Y -667.654,Z 408.457,A 0.000,B 0.000,C 90.000,E1 298.359} C_DIS
LIN {X 0.249,Y -669.466,Z 408.453,A 0.000,B 0.000,C 90.000,E1 297.590} C_DIS
LIN {X -0.071,Y -673.198,Z 408.444,A 0.000,B 0.000,C 90.000,E1 295.924} C_DIS
LIN {X 0.030,Y -675.201,Z 408.439,A 0.000,B 0.000,C 90.000,E1 294.951} C_DIS
LIN {X -0.139,Y -677.201,Z 408.433,A 0.000,B 0.000,C 90.000,E1 294.003} C_DIS
LIN {X 0.257,Y -679.027,Z 408.427,A 0.000,B 0.000,C 90.000,E1 292.770} C_DIS
LIN {X -0.128,Y -680.009,Z 408.421,A 0.000,B 0.000,C 90.000,E1 291.844} C_DIS
LIN {X 0.134,Y -680.653,Z 408.416,A 0.000,B 0.000,C 90.000,E1 290.865} C_DIS
LIN {X -0.183,Y -681.029,Z 408.412,A 0.000,B 0.000,C 90.000,E1 290.174} C_DIS
LIN {X -0.097,Y -681.209,Z 408.408,A 0.000,B 0.000,C 90.000,E1 289.450} C_DIS
LIN {X -0.005,Y -681.198,Z 408.404,A 0.000,B 0.000,C 90.000,E1 288.725} C_DIS
LIN {X 0.087,Y -681.093,Z 408.400,A 0.000,B 0.000,C 90.000,E1 288.000} C_DIS
LIN {X 0.101,Y -680.614,Z 408.393,A 0.000,B 0.000,C 90.000,E1 286.804} C_DIS
LIN {X 0.108,Y -679.863,Z 408.387,A 0.000,B 0.000,C 90.000,E1 285.607} C_DIS
LIN {X 0.035,Y -679.573,Z 408.384,A 0.000,B 0.000,C 90.000,E1 285.134} C_DIS
LIN {X -0.075,Y -678.110,Z 408.375,A 0.000,B 0.000,C 90.000,E1 283.467} C_DIS
LIN {X -0.359,Y -677.413,Z 408.371,A 0.000,B 0.000,C 90.000,E1 282.771} C_DIS
LIN {X 0.118,Y -676.449,Z 408.366,A 0.000,B 0.000,C 90.000,E1 281.771} C_DIS
LIN {X 0.094,Y -674.168,Z 408.355,A 0.000,B 0.000,C 90.000,E1 279.849} C_DIS
LIN {X -0.169,Y -671.826,Z 408.343,A 0.000,B 0.000,C 90.000,E1 277.701} C_DIS
LIN {X -0.008,Y -669.726,Z 408.331,A 0.000,B 0.000,C 90.000,E1 275.511} C_DIS
LIN {X -0.307,Y -668.117,Z 408.321,A 0.000,B 0.000,C 90.000,E1 273.841} C_DIS
LIN {X -0.248,Y -667.206,Z 408.316,A 0.000,B 0.000,C 90.000,E1 272.865} C_DIS
LIN {X 0.133,Y -665.847,Z 408.308,A 0.000,B 0.000,C 90.000,E1 271.375} C_DIS
LIN {X -0.195,Y -665.376,Z 408.305,A 0.000,B 0.000,C 90.000,E1 270.917} C_DIS
LIN {X 0.305,Y -663.917,Z 408.298,A 0.000,B 0.000,C 90.000,E1 269.656} C_DIS
LIN {X 0.288,Y -662.465,Z 408.293,A 0.000,B 0.000,C 90.000,E1 268.682} C_DIS
LIN {X 0.114,Y -662.001,Z 408.292,A 0.000,B 0.000,C 90.000,E1 268.453} C_DIS
LIN {X -0.062,Y -661.703,Z 408.290,A 0.000,B 0.000,C 90.000,E1 268.224} C_DIS
LIN {X -0.216,Y -661.269,Z 408.289,A 0.000,B 0.000,C 90.000,E1 267.993} C_DIS
LIN {X 0.268,Y -661.018,Z 408.287,A 0.000,B 0.000,C 90.000,E1 267.707} C_DIS
LIN {X -0.091,Y -660.169,Z 408.285,A 0.000,B 0.000,C 90.000,E1 267.249} C_DIS
LIN {X 0.237,Y -659.422,Z 408.282,A 0.000,B 0.000,C 90.000,E1 266.731} C_DIS
LIN {X -0.008,Y -657.100,Z 408.275,A 0.000,B 0.000,C 90.000,E1 265.527} C_DIS
LIN {X 0.104,Y -655.471,Z 408.271,A 0.000,B 0.000,C 90.000,E1 264.780} C_DIS
LIN {X 0.055,Y -653.173,Z 408.266,A 0.000,B 0.000,C 90.000,E1 263.799} C_DIS
LIN {X -0.250,Y -649.916,Z 408.259,A 0.000,B 0.000,C 90.000,E1 262.591} C_DIS
LIN {X 0.110,Y -646.531,Z 408.252,A 0.000,B 0.000,C 90.000,E1 261.319} C_DIS
LIN {X 0.188,Y -644.298,Z 408.248,A 0.000,B 0.000,C 90.000,E1 260.566} C_DIS
LIN {X -0.240,Y -639.803,Z 408.239,A 0.000,B 0.000,C 90.000,E1 259.106} C_DIS
LIN {X 0.351,Y -636.750,Z 408.234,A 0.000,B 0.000,C 90.000,E1 258.049} C_DIS
LIN {X -0.221,Y -631.980,Z 408.225,A 0.000,B 0.000,C 90.000,E1 256.589} C_DIS
LIN {X 0.213,Y -627.762,Z 408.218,A 0.000,B 0.000,C 90.000,E1 255.283} C_DIS
LIN {X -0.233,Y -622.398,Z 408.210,A 0.000,B 0.000,C 90.000,E1 253.795} C_DIS
LIN {X 0.033,Y -617.754,Z 408.203,A 0.000,B 0.000,C 90.000,E1 252.489} C_DIS
LIN {X -0.191,Y -612.999,Z 408.196,A 0.000,B 0.000,C 90.000,E1 251.221} C_DIS
LIN {X 0.284,Y -608.027,Z 408.188,A 0.000,B 0.000,C 90.000,E1 249.880} C_DIS
LIN {X 0.104,Y -602.895,Z 408.181,A 0.000,B 0.000,C 90.000,E1 248.592} C_DIS
LIN {X 0.144,Y -598.653,Z 408.175,A 0.000,B 0.000,C 90.000,E1 247.539} C_DIS
LIN {X 0.033,Y -593.180,Z 408.168,A 0.000,B 0.000,C 90.000,E1 246.230} C_DIS
LIN {X -0.174,Y -587.664,Z 408.161,A 0.000,B 0.000,C 90.000,E1 244.921} C_DIS
LIN {X 0.286,Y -579.824,Z 408.150,A 0.000,B 0.000,C 90.000,E1 242.999} C_DIS
LIN {X 0.194,Y -573.119,Z 408.141,A 0.000,B 0.000,C 90.000,E1 241.385} C_DIS
LIN {X -0.077,Y -567.698,Z 408.134,A 0.000,B 0.000,C 90.000,E1 240.049} C_DIS
LIN {X -0.180,Y -558.238,Z 408.120,A 0.000,B 0.000,C 90.000,E1 237.582} C_DIS
LIN {X -0.002,Y -549.302,Z 408.106,A 0.000,B 0.000,C 90.000,E1 235.055} C_DIS
LIN {X -0.008,Y -542.574,Z 408.095,A 0.000,B 0.000,C 90.000,E1 233.084} C_DIS
LIN {X 0.018,Y -537.748,Z 408.087,A 0.000,B 0.000,C 90.000,E1 231.662} C_DIS
LIN {X -0.036,Y -531.013,Z 408.076,A 0.000,B 0.000,C 90.000,E1 229.666} C_DIS
LIN {X -0.053,Y -522.876,Z 408.061,A 0.000,B 0.000,C 90.000,E1 227.067} C_DIS
LIN {X -0.030,Y -518.492,Z 408.053,A 0.000,B 0.000,C 90.000,E1 225.607} C_DIS
LIN {X -0.197,Y -513.340,Z 408.044,A 0.000,B 0.000,C 90.000,E1 223.866} C_DIS
LIN {X -0.093,Y -508.227,Z 408.034,A 0.000,B 0.000,C 90.000,E1 222.081} C_DIS
LIN {X -0.107,Y -503.305,Z 408.024,A 0.000,B 0.000,C 90.000,E1 220.297} C_DIS
LIN {X 0.078,Y -497.745,Z 408.012,A 0.000,B 0.000,C 90.000,E1 218.177} C_DIS
LIN {X -0.033,Y -493.150,Z 408.002,A 0.000,B 0.000,C 90.000,E1 216.377} C_DIS
LIN {X -0.020,Y -487.937,Z 407.990,A 0.000,B 0.000,C 90.000,E1 214.246} C_DIS
LIN {X -0.106,Y -483.651,Z 407.980,A 0.000,B 0.000,C 90.000,E1 212.418} C_DIS
LIN {X 0.129,Y -479.377,Z 407.970,A 0.000,B 0.000,C 90.000,E1 210.541} C_DIS
LIN {X 0.023,Y -475.128,Z 407.959,A 0.000,B 0.000,C 90.000,E1 208.693} C_DIS
LIN {X -0.114,Y -472.230,Z 407.953,A 0.000,B 0.000,C 90.000,E1 207.462} C_DIS
LIN {X 0.127,Y -469.297,Z 407.946,A 0.000,B 0.000,C 90.000,E1 206.181} C_DIS
LIN {X -0.166,Y -465.527,Z 407.937,A 0.000,B 0.000,C 90.000,E1 204.643} C_DIS
LIN {X 0.191,Y -462.502,Z 407.930,A 0.000,B 0.000,C 90.000,E1 203.334} C_DIS
LIN {X 0.244,Y -457.162,Z 407.917,A 0.000,B 0.000,C 90.000,E1 201.099} C_DIS
LIN {X 0.145,Y -451.459,Z 407.903,A 0.000,B 0.000,C 90.000,E1 198.544} C_DIS
LIN {X 0.027,Y -446.318,Z 407.889,A 0.000,B 0.000,C 90.000,E1 195.969} C_DIS
LIN {X -0.096,Y -442.239,Z 407.876,A 0.000,B 0.000,C 90.000,E1 193.703} C_DIS
LIN {X -0.217,Y -438.411,Z 407.863,A 0.000,B 0.000,C 90.000,E1 191.422} C_DIS
LIN {X 0.052,Y -434.391,Z 407.849,A 0.000,B 0.000,C 90.000,E1 188.746} C_DIS
LIN {X -0.113,Y -431.692,Z 407.838,A 0.000,B 0.000,C 90.000,E1 186.777} C_DIS
LIN {X 0.155,Y -428.508,Z 407.823,A 0.000,B 0.000,C 90.000,E1 184.073} C_DIS
LIN {X -0.138,Y -425.913,Z 407.808,A 0.000,B 0.000,C 90.000,E1 181.432} C_DIS
LIN {X 0.035,Y -423.406,Z 407.787,A 0.000,B 0.000,C 90.000,E1 177.707} C_DIS
LIN {X 0.134,Y -422.360,Z 407.769,A 0.000,B 0.000,C 90.000,E1 174.318} C_DIS
LIN {X 0.127,Y -422.518,Z 407.744,A 0.000,B 0.000,C 90.000,E1 169.926} C_DIS
LIN {X -0.075,Y -423.430,Z 407.731,A 0.000,B 0.000,C 90.000,E1 167.589} C_DIS
LIN {X 0.127,Y -425.130,Z 407.716,A 0.000,B 0.000,C 90.000,E1 164.866} C_DIS
LIN {X 0.098,Y -428.129,Z 407.697,A 0.000,B 0.000,C 90.000,E1 161.511} C_DIS
LIN {X -0.199,Y -430.821,Z 407.684,A 0.000,B 0.000,C 90.000,E1 159.209} C_DIS
LIN {X 0.045,Y -433.976,Z 407.671,A 0.000,B 0.000,C 90.000,E1 156.847} C_DIS
LIN {X 0.081,Y -439.864,Z 407.651,A 0.000,B 0.000,C 90.000,E1 153.204} C_DIS
LIN {X -0.022,Y -446.904,Z 407.631,A 0.000,B 0.000,C 90.000,E1 149.616} C_DIS
LIN {X 0.121,Y -452.099,Z 407.619,A 0.000,B 0.000,C 90.000,E1 147.327} C_DIS
LIN {X 0.006,Y -458.688,Z 407.604,A 0.000,B 0.000,C 90.000,E1 144.769} C_DIS
LIN {X 0.024,Y -466.973,Z 407.588,A 0.000,B 0.000,C 90.000,E1 141.904} C_DIS
LIN {X -0.114,Y -475.858,Z 407.573,A 0.000,B 0.000,C 90.000,E1 139.094} C_DIS
LIN {X -0.015,Y -479.735,Z 407.566,A 0.000,B 0.000,C 90.000,E1 137.838} C_DIS
LIN {X -0.180,Y -483.470,Z 407.559,A 0.000,B 0.000,C 90.000,E1 136.620} C_DIS
LIN {X 0.036,Y -487.004,Z 407.552,A 0.000,B 0.000,C 90.000,E1 135.364} C_DIS
LIN {X -0.009,Y -488.700,Z 407.549,A 0.000,B 0.000,C 90.000,E1 134.757} C_DIS
LIN {X -0.062,Y -491.650,Z 407.542,A 0.000,B 0.000,C 90.000,E1 133.542} C_DIS
LIN {X -0.048,Y -494.417,Z 407.535,A 0.000,B 0.000,C 90.000,E1 132.324} C_DIS
LIN {X 0.159,Y -496.130,Z 407.530,A 0.000,B 0.000,C 90.000,E1 131.391} C_DIS
LIN {X 0.059,Y -497.486,Z 407.525,A 0.000,B 0.000,C 90.000,E1 130.496} C_DIS
LIN {X 0.294,Y -498.558,Z 407.520,A 0.000,B 0.000,C 90.000,E1 129.564} C_DIS
LIN {X -0.095,Y -499.185,Z 407.515,A 0.000,B 0.000,C 90.000,E1 128.705} C_DIS
LIN {X 0.088,Y -499.296,Z 407.513,A 0.000,B 0.000,C 90.000,E1 128.382} C_DIS
LIN {X -0.290,Y -499.165,Z 407.508,A 0.000,B 0.000,C 90.000,E1 127.523} C_DIS
LIN {X 0.158,Y -498.756,Z 407.505,A 0.000,B 0.000,C 90.000,E1 126.870} C_DIS
LIN {X -0.224,Y -497.783,Z 407.500,A 0.000,B 0.000,C 90.000,E1 126.011} C_DIS
LIN {X -0.214,Y -496.465,Z 407.495,A 0.000,B 0.000,C 90.000,E1 125.105} C_DIS
LIN {X -0.077,Y -495.401,Z 407.492,A 0.000,B 0.000,C 90.000,E1 124.485} C_DIS
LIN {X 0.053,Y -494.058,Z 407.488,A 0.000,B 0.000,C 90.000,E1 123.865} C_DIS
LIN {X 0.023,Y -491.832,Z 407.483,A 0.000,B 0.000,C 90.000,E1 122.959} C_DIS
LIN {X -0.040,Y -489.085,Z 407.478,A 0.000,B 0.000,C 90.000,E1 122.054} C_DIS
LIN {X 0.021,Y -485.944,Z 407.473,A 0.000,B 0.000,C 90.000,E1 121.131} C_DIS
LIN {X 0.051,Y -482.516,Z 407.468,A 0.000,B 0.000,C 90.000,E1 120.207} C_DIS
LIN {X -0.180,Y -478.051,Z 407.462,A 0.000,B 0.000,C 90.000,E1 119.155} C_DIS
LIN {X -0.063,Y -472.724,Z 407.455,A 0.000,B 0.000,C 90.000,E1 117.897} C_DIS
LIN {X 0.161,Y -466.953,Z 407.448,A 0.000,B 0.000,C 90.000,E1 116.616} C_DIS
LIN {X 0.128,Y -458.049,Z 407.437,A 0.000,B 0.000,C 90.000,E1 114.719} C_DIS
LIN {X -0.145,Y -449.282,Z 407.427,A 0.000,B 0.000,C 90.000,E1 112.898} C_DIS
LIN {X -0.185,Y -449.288,Z 407.427,A 0.000,B 0.000,C 90.000,E1 112.898} C_DIS
LIN {X -0.107,Y -457.390,Z 407.410,A 0.000,B 0.000,C 90.000,E1 109.758} C_DIS
LIN {X -0.023,Y -466.027,Z 407.387,A 0.000,B 0.000,C 90.000,E1 105.607} C_DIS
LIN {X 0.151,Y -467.594,Z 407.383,A 0.000,B 0.000,C 90.000,E1 104.954} C_DIS
LIN {X -0.116,Y -468.592,Z 407.380,A 0.000,B 0.000,C 90.000,E1 104.356} C_DIS
LIN {X 0.110,Y -475.823,Z 407.357,A 0.000,B 0.000,C 90.000,E1 100.254} C_DIS
LIN {X -0.053,Y -476.315,Z 407.355,A 0.000,B 0.000,C 90.000,E1 99.962} C_DIS
LIN {X -0.105,Y -481.806,Z 407.331,A 0.000,B 0.000,C 90.000,E1 95.625} C_DIS
LIN {X 0.221,Y -482.175,Z 407.330,A 0.000,B 0.000,C 90.000,E1 95.277} C_DIS
LIN {X 0.156,Y -485.319,Z 407.306,A 0.000,B 0.000,C 90.000,E1 90.974} C_DIS
LIN {X -0.019,Y -485.536,Z 407.304,A 0.000,B 0.000,C 90.000,E1 90.688} C_DIS
LIN {X 0.188,Y -486.324,Z 407.282,A 0.000,B 0.000,C 90.000,E1 86.674} C_DIS
LIN {X -0.162,Y -486.298,Z 407.278,A 0.000,B 0.000,C 90.000,E1 86.102} C_DIS
LIN {X 0.042,Y -484.696,Z 407.254,A 0.000,B 0.000,C 90.000,E1 81.781} C_DIS
LIN {X -0.090,Y -484.588,Z 407.253,A 0.000,B 0.000,C 90.000,E1 81.489} C_DIS
LIN {X -0.210,Y -480.524,Z 407.227,A 0.000,B 0.000,C 90.000,E1 76.881} C_DIS
LIN {X 0.155,Y -474.275,Z 407.201,A 0.000,B 0.000,C 90.000,E1 72.181} C_DIS
LIN {X 0.122,Y -473.827,Z 407.199,A 0.000,B 0.000,C 90.000,E1 71.873} C_DIS
LIN {X 0.072,Y -469.277,Z 407.186,A 0.000,B 0.000,C 90.000,E1 69.464} C_DIS
LIN {X 0.195,Y -469.308,Z 407.186,A 0.000,B 0.000,C 90.000,E1 69.444} C_DIS
LIN {X -0.192,Y -479.437,Z 407.179,A 0.000,B 0.000,C 90.000,E1 68.156} C_DIS
LIN {X -0.196,Y -488.818,Z 407.172,A 0.000,B 0.000,C 90.000,E1 66.922} C_DIS
LIN {X 0.097,Y -494.555,Z 407.167,A 0.000,B 0.000,C 90.000,E1 66.125} C_DIS
LIN {X 0.063,Y -503.241,Z 407.161,A 0.000,B 0.000,C 90.000,E1 64.921} C_DIS
LIN {X 0.066,Y -509.199,Z 407.156,A 0.000,B 0.000,C 90.000,E1 64.024} C_DIS
LIN {X -0.022,Y -512.025,Z 407.153,A 0.000,B 0.000,C 90.000,E1 63.589} C_DIS
LIN {X -0.038,Y -515.553,Z 407.150,A 0.000,B 0.000,C 90.000,E1 62.999} C_DIS
LIN {X -0.024,Y -518.822,Z 407.147,A 0.000,B 0.000,C 90.000,E1 62.410} C_DIS
LIN {X 0.016,Y -521.846,Z 407.143,A 0.000,B 0.000,C 90.000,E1 61.820} C_DIS
LIN {X -0.171,Y -524.630,Z 407.140,A 0.000,B 0.000,C 90.000,E1 61.257} C_DIS
LIN {X -0.089,Y -527.110,Z 407.137,A 0.000,B 0.000,C 90.000,E1 60.667} C_DIS
LIN {X 0.008,Y -529.365,Z 407.134,A 0.000,B 0.000,C 90.000,E1 60.078} C_DIS
LIN {X 0.119,Y -531.423,Z 407.131,A 0.000,B 0.000,C 90.000,E1 59.488} C_DIS
LIN {X 0.063,Y -533.177,Z 407.127,A 0.000,B 0.000,C 90.000,E1 58.918} C_DIS
LIN {X 0.204,Y -534.734,Z 407.124,A 0.000,B 0.000,C 90.000,E1 58.329} C_DIS
LIN {X -0.091,Y -535.478,Z 407.123,A 0.000,B 0.000,C 90.000,E1 58.074} C_DIS
LIN {X 0.056,Y -537.135,Z 407.118,A 0.000,B 0.000,C 90.000,E1 57.199} C_DIS
LIN {X 0.067,Y -538.321,Z 407.113,A 0.000,B 0.000,C 90.000,E1 56.342} C_DIS
LIN {X -0.214,Y -538.892,Z 407.110,A 0.000,B 0.000,C 90.000,E1 55.801} C_DIS
LIN {X 0.271,Y -539.389,Z 407.105,A 0.000,B 0.000,C 90.000,E1 54.895} C_DIS
LIN {X 0.005,Y -539.515,Z 407.100,A 0.000,B 0.000,C 90.000,E1 54.069} C_DIS
LIN {X 0.056,Y -539.268,Z 407.096,A 0.000,B 0.000,C 90.000,E1 53.210} C_DIS
LIN {X 0.104,Y -538.770,Z 407.091,A 0.000,B 0.000,C 90.000,E1 52.351} C_DIS
LIN {X -0.267,Y -537.755,Z 407.085,A 0.000,B 0.000,C 90.000,E1 51.251} C_DIS
LIN {X 0.101,Y -536.826,Z 407.080,A 0.000,B 0.000,C 90.000,E1 50.356} C_DIS
LIN {X 0.050,Y -535.424,Z 407.074,A 0.000,B 0.000,C 90.000,E1 49.218} C_DIS
LIN {X -0.011,Y -534.218,Z 407.069,A 0.000,B 0.000,C 90.000,E1 48.366} C_DIS
LIN {X -0.120,Y -532.117,Z 407.061,A 0.000,B 0.000,C 90.000,E1 46.944} C_DIS
LIN {X 0.024,Y -529.574,Z 407.051,A 0.000,B 0.000,C 90.000,E1 45.202} C_DIS
LIN {X 0.112,Y -527.184,Z 407.042,A 0.000,B 0.000,C 90.000,E1 43.461} C_DIS
LIN {X 0.231,Y -525.380,Z 407.034,A 0.000,B 0.000,C 90.000,E1 42.000} C_DIS
LIN {X -0.126,Y -523.212,Z 407.024,A 0.000,B 0.000,C 90.000,E1 40.297} C_DIS
LIN {X -0.020,Y -521.494,Z 407.016,A 0.000,B 0.000,C 90.000,E1 38.830} C_DIS
LIN {X 0.055,Y -519.718,Z 407.008,A 0.000,B 0.000,C 90.000,E1 37.363} C_DIS
LIN {X 0.137,Y -517.495,Z 406.998,A 0.000,B 0.000,C 90.000,E1 35.598} C_DIS
LIN {X -0.118,Y -516.013,Z 406.991,A 0.000,B 0.000,C 90.000,E1 34.452} C_DIS
LIN {X 0.012,Y -513.625,Z 406.982,A 0.000,B 0.000,C 90.000,E1 32.673} C_DIS
LIN {X -0.184,Y -511.253,Z 406.972,A 0.000,B 0.000,C 90.000,E1 30.924} C_DIS
LIN {X -0.032,Y -508.150,Z 406.959,A 0.000,B 0.000,C 90.000,E1 28.537} C_DIS
LIN {X -0.016,Y -505.300,Z 406.945,A 0.000,B 0.000,C 90.000,E1 26.155} C_DIS
LIN {X -0.058,Y -502.711,Z 406.932,A 0.000,B 0.000,C 90.000,E1 23.770} C_DIS
LIN {X 0.102,Y -500.531,Z 406.919,A 0.000,B 0.000,C 90.000,E1 21.354} C_DIS
LIN {X -0.092,Y -498.540,Z 406.904,A 0.000,B 0.000,C 90.000,E1 18.671} C_DIS
LIN {X 0.040,Y -497.521,Z 406.895,A 0.000,B 0.000,C 90.000,E1 17.149} C_DIS
LIN {X -0.149,Y -496.533,Z 406.887,A 0.000,B 0.000,C 90.000,E1 15.662} C_DIS
LIN {X -0.057,Y -495.312,Z 406.875,A 0.000,B 0.000,C 90.000,E1 13.536} C_DIS
LIN {X 0.194,Y -494.203,Z 406.860,A 0.000,B 0.000,C 90.000,E1 10.782} C_DIS
LIN {X -0.141,Y -493.735,Z 406.840,A 0.000,B 0.000,C 90.000,E1 7.182} C_DIS
LIN {X 0.172,Y -494.100,Z 406.825,A 0.000,B 0.000,C 90.000,E1 4.416} C_DIS
LIN {X -0.242,Y -494.365,Z 406.820,A 0.000,B 0.000,C 90.000,E1 3.555} C_DIS
LIN {X 0.048,Y -495.192,Z 406.811,A 0.000,B 0.000,C 90.000,E1 2.007} C_DIS
LIN {X -0.101,Y -498.619,Z 406.789,A 0.000,B 0.000,C 90.000,E1 357.993} C_DIS
LIN {X 0.090,Y -502.931,Z 406.770,A 0.000,B 0.000,C 90.000,E1 354.666} C_DIS
LIN {X -0.068,Y -506.121,Z 406.759,A 0.000,B 0.000,C 90.000,E1 352.591} C_DIS
LIN {X -0.038,Y -510.344,Z 406.746,A 0.000,B 0.000,C 90.000,E1 350.208} C_DIS
LIN {X 0.174,Y -517.258,Z 406.728,A 0.000,B 0.000,C 90.000,E1 346.937} C_DIS
LIN {X -0.135,Y -522.976,Z 406.715,A 0.000,B 0.000,C 90.000,E1 344.629} C_DIS
LIN {X -0.157,Y -528.213,Z 406.703,A 0.000,B 0.000,C 90.000,E1 342.598} C_DIS
LIN {X 0.111,Y -533.572,Z 406.692,A 0.000,B 0.000,C 90.000,E1 340.550} C_DIS
LIN {X 0.183,Y -539.167,Z 406.681,A 0.000,B 0.000,C 90.000,E1 338.539} C_DIS
LIN {X 0.060,Y -544.039,Z 406.671,A 0.000,B 0.000,C 90.000,E1 336.847} C_DIS
LIN {X -0.181,Y -547.365,Z 406.665,A 0.000,B 0.000,C 90.000,E1 335.741} C_DIS
LIN {X -0.126,Y -553.270,Z 406.654,A 0.000,B 0.000,C 90.000,E1 333.768} C_DIS
LIN {X -0.156,Y -559.456,Z 406.643,A 0.000,B 0.000,C 90.000,E1 331.820} C_DIS
LIN {X 0.079,Y -563.905,Z 406.636,A 0.000,B 0.000,C 90.000,E1 330.411} C_DIS
LIN {X -0.213,Y -569.366,Z 406.627,A 0.000,B 0.000,C 90.000,E1 328.791} C_DIS
LIN {X 0.277,Y -573.796,Z 406.619,A 0.000,B 0.000,C 90.000,E1 327.375} C_DIS
LIN {X -0.285,Y -579.129,Z 406.610,A 0.000,B 0.000,C 90.000,E1 325.801} C_DIS
LIN {X 0.055,Y -584.443,Z 406.601,A 0.000,B 0.000,C 90.000,E1 324.149} C_DIS
LIN {X -0.100,Y -589.896,Z 406.592,A 0.000,B 0.000,C 90.000,E1 322.557} C_DIS
LIN {X -0.157,Y -597.339,Z 406.580,A 0.000,B 0.000,C 90.000,E1 320.436} C_DIS
LIN {X 0.089,Y -602.031,Z 406.573,A 0.000,B 0.000,C 90.000,E1 319.094} C_DIS
